   t1[18698] := -0.0536004;
   t1[18699] := -0.0617994;
   t1[18700] := 0.3399203;
   t1[18701] := 0.3337824;
   t1[18702] := 0.3265423;
   t1[18703] := 0.3181666;
   t1[18704] := 0.3086217;
   t1[18705] := 0.2978742;
   t1[18706] := 0.2858903;
   t1[18707] := 0.2726368;
   t1[18708] := 0.2580868;
   t1[18709] := 0.2423165;
   t1[18710] := 0.2254834;
   t1[18711] := 0.2077472;
   t1[18712] := 0.1892676;
   t1[18713] := 0.1702043;
   t1[18714] := 0.1507169;
   t1[18715] := 0.1309651;
   t1[18716] := 0.1111085;
   t1[18717] := 0.091307;
   t1[18718] := 0.0717201;
   t1[18719] := 0.0525076;
   t1[18720] := 0.033829;
   t1[18721] := 0.0158441;
   t1[18722] := -0.0012874;
   t1[18723] := -0.0174059;
   t1[18724] := -0.0323517;
   t1[18725] := -0.045965;
   t1[18726] := -0.0580863;
   t1[18727] := -0.0685566;
   t1[18728] := -0.0773026;
   t1[18729] := -0.084413;
   t1[18730] := -0.0899949;
   t1[18731] := -0.0941551;
   t1[18732] := -0.0970005;
   t1[18733] := -0.0986381;
   t1[18734] := -0.0991749;
   t1[18735] := -0.0987177;
   t1[18736] := -0.0973734;
   t1[18737] := -0.095249;
   t1[18738] := -0.0924515;
   t1[18739] := -0.0890877;
   t1[18740] := -0.0852646;
   t1[18741] := -0.0810891;
   t1[18742] := -0.0766682;
   t1[18743] := -0.0721086;
   t1[18744] := -0.0675175;
   t1[18745] := -0.0630017;
   t1[18746] := -0.0586682;
   t1[18747] := -0.0546078;
   t1[18748] := -0.0508318;
   t1[18749] := -0.0473261;
   t1[18750] := 0.1759748;
   t1[18751] := 0.1774203;
   t1[18752] := 0.1786771;
   t1[18753] := 0.1797362;
   t1[18754] := 0.1805886;
   t1[18755] := 0.1812253;
   t1[18756] := 0.1816373;
   t1[18757] := 0.1818157;
   t1[18758] := 0.1817521;
   t1[18759] := 0.1814474;
   t1[18760] := 0.1809096;
   t1[18761] := 0.1801469;
   t1[18762] := 0.1791678;
   t1[18763] := 0.1779805;
   t1[18764] := 0.1765932;
   t1[18765] := 0.1750143;
   t1[18766] := 0.173252;
   t1[18767] := 0.1713147;
   t1[18768] := 0.1692105;
   t1[18769] := 0.1669478;
   t1[18770] := 0.1645349;
   t1[18771] := 0.1619801;
   t1[18772] := 0.1592916;
   t1[18773] := 0.1564777;
   t1[18774] := 0.1535467;
   t1[18775] := 0.1505069;
   t1[18776] := 0.1473666;
   t1[18777] := 0.1441341;
   t1[18778] := 0.1408151;
   t1[18779] := 0.1374107;
   t1[18780] := 0.1339216;
   t1[18781] := 0.1303483;
   t1[18782] := 0.1266915;
   t1[18783] := 0.1229517;
   t1[18784] := 0.1191295;
   t1[18785] := 0.1152255;
   t1[18786] := 0.1112403;
   t1[18787] := 0.1071746;
   t1[18788] := 0.1030288;
   t1[18789] := 0.0988036;
   t1[18790] := 0.0944996;
   t1[18791] := 0.0901174;
   t1[18792] := 0.0856576;
   t1[18793] := 0.0811207;
   t1[18794] := 0.0765074;
   t1[18795] := 0.0718182;
   t1[18796] := 0.0670538;
   t1[18797] := 0.062218;
   t1[18798] := 0.057331;
   t1[18799] := 0.0524179;
   t1[18800] := 0.2070498;
   t1[18801] := 0.1995114;
   t1[18802] := 0.1919864;
   t1[18803] := 0.1845329;
   t1[18804] := 0.1772084;
   t1[18805] := 0.1700709;
   t1[18806] := 0.1631781;
   t1[18807] := 0.156588;
   t1[18808] := 0.1503544;
   t1[18809] := 0.1444713;
   t1[18810] := 0.1388855;
   t1[18811] := 0.1335424;
   t1[18812] := 0.1283877;
   t1[18813] := 0.1233668;
   t1[18814] := 0.1184252;
   t1[18815] := 0.1135085;
   t1[18816] := 0.1085621;
   t1[18817] := 0.1035315;
   t1[18818] := 0.0983623;
   t1[18819] := 0.0929999;
   t1[18820] := 0.0873899;
   t1[18821] := 0.0814778;
   t1[18822] := 0.0752091;
   t1[18823] := 0.0685292;
   t1[18824] := 0.0613837;
   t1[18825] := 0.0537182;
   t1[18826] := 0.045478;
   t1[18827] := 0.0366092;
   t1[18828] := 0.0271076;
   t1[18829] := 0.0170635;
   t1[18830] := 0.0065778;
   t1[18831] := -0.0042485;
   t1[18832] := -0.0153147;
   t1[18833] := -0.0265199;
   t1[18834] := -0.037763;
   t1[18835] := -0.0489433;
   t1[18836] := -0.0599599;
   t1[18837] := -0.0707118;
   t1[18838] := -0.0810982;
   t1[18839] := -0.0910181;
   t1[18840] := -0.1003708;
   t1[18841] := -0.1090552;
   t1[18842] := -0.1169706;
   t1[18843] := -0.124016;
   t1[18844] := -0.1300905;
   t1[18845] := -0.1350932;
   t1[18846] := -0.1389232;
   t1[18847] := -0.1415044;
   t1[18848] := -0.1428838;
   t1[18849] := -0.1431469;
   t1[18850] := 0.2326834;
   t1[18851] := 0.2246485;
   t1[18852] := 0.2165409;
   t1[18853] := 0.208421;
   t1[18854] := 0.2003494;
   t1[18855] := 0.1923865;
   t1[18856] := 0.1845929;
   t1[18857] := 0.177029;
   t1[18858] := 0.1697522;
   t1[18859] := 0.162768;
   t1[18860] := 0.1560417;
   t1[18861] := 0.1495374;
   t1[18862] := 0.1432192;
   t1[18863] := 0.1370513;
   t1[18864] := 0.1309978;
   t1[18865] := 0.1250227;
   t1[18866] := 0.1190902;
   t1[18867] := 0.1131645;
   t1[18868] := 0.1072096;
   t1[18869] := 0.1011897;
   t1[18870] := 0.0950688;
   t1[18871] := 0.0888111;
   t1[18872] := 0.0823807;
   t1[18873] := 0.0757418;
   t1[18874] := 0.0688584;
   t1[18875] := 0.0616946;
   t1[18876] := 0.0542147;
   t1[18877] := 0.0463829;
   t1[18878] := 0.0381994;
   t1[18879] := 0.0297315;
   t1[18880] := 0.0210542;
   t1[18881] := 0.0122423;
   t1[18882] := 0.0033709;
   t1[18883] := -0.0054852;
   t1[18884] := -0.014251;
   t1[18885] := -0.0228515;
   t1[18886] := -0.0312118;
   t1[18887] := -0.0392571;
   t1[18888] := -0.0469123;
   t1[18889] := -0.0541025;
   t1[18890] := -0.0607528;
   t1[18891] := -0.0667883;
   t1[18892] := -0.072134;
   t1[18893] := -0.076715;
   t1[18894] := -0.0804563;
   t1[18895] := -0.0832831;
   t1[18896] := -0.0851203;
   t1[18897] := -0.0859139;
   t1[18898] := -0.0857146;
   t1[18899] := -0.0846053;
   t1[18900] := 0.0673334;
   t1[18901] := 0.0664519;
   t1[18902] := 0.0653818;
   t1[18903] := 0.0641012;
   t1[18904] := 0.0625887;
   t1[18905] := 0.0608225;
   t1[18906] := 0.0587809;
   t1[18907] := 0.0564422;
   t1[18908] := 0.0537876;
   t1[18909] := 0.0508431;
   t1[18910] := 0.0476698;
   t1[18911] := 0.0443297;
   t1[18912] := 0.0408848;
   t1[18913] := 0.0373974;
   t1[18914] := 0.0339294;
   t1[18915] := 0.0305429;
   t1[18916] := 0.0272999;
   t1[18917] := 0.0242625;
   t1[18918] := 0.0214929;
   t1[18919] := 0.019053;
   t1[18920] := 0.0170049;
   t1[18921] := 0.0154107;
   t1[18922] := 0.0143324;
   t1[18923] := 0.0138322;
   t1[18924] := 0.013972;
   t1[18925] := 0.0148139;
   t1[18926] := 0.0164201;
   t1[18927] := 0.0188521;
   t1[18928] := 0.022123;
   t1[18929] := 0.0261538;
   t1[18930] := 0.0308553;
   t1[18931] := 0.0361382;
   t1[18932] := 0.0419132;
   t1[18933] := 0.0480911;
   t1[18934] := 0.0545826;
   t1[18935] := 0.0612985;
   t1[18936] := 0.0681495;
   t1[18937] := 0.0750462;
   t1[18938] := 0.0818996;
   t1[18939] := 0.0886203;
   t1[18940] := 0.095119;
   t1[18941] := 0.1013065;
   t1[18942] := 0.1070935;
   t1[18943] := 0.1123908;
   t1[18944] := 0.1171091;
   t1[18945] := 0.1211592;
   t1[18946] := 0.1244517;
   t1[18947] := 0.1269166;
   t1[18948] := 0.1285797;
   t1[18949] := 0.1294967;
   t1[18950] := 0.0280284;
   t1[18951] := 0.0228271;
   t1[18952] := 0.0181762;
   t1[18953] := 0.0141364;
   t1[18954] := 0.0107684;
   t1[18955] := 0.0081328;
   t1[18956] := 0.0062904;
   t1[18957] := 0.0053019;
   t1[18958] := 0.0052228;
   t1[18959] := 0.0060285;
   t1[18960] := 0.0076314;
   t1[18961] := 0.0099423;
   t1[18962] := 0.0128719;
   t1[18963] := 0.0163309;
   t1[18964] := 0.02023;
   t1[18965] := 0.0244799;
   t1[18966] := 0.0289914;
   t1[18967] := 0.0336752;
   t1[18968] := 0.0384419;
   t1[18969] := 0.0432023;
   t1[18970] := 0.0478672;
   t1[18971] := 0.0523472;
   t1[18972] := 0.056553;
   t1[18973] := 0.0603954;
   t1[18974] := 0.0637852;
   t1[18975] := 0.0666328;
   t1[18976] := 0.0688493;
   t1[18977] := 0.0703455;
   t1[18978] := 0.0710739;
   t1[18979] := 0.0710653;
   t1[18980] := 0.070359;
   t1[18981] := 0.0689945;
   t1[18982] := 0.0670113;
   t1[18983] := 0.0644488;
   t1[18984] := 0.0613464;
   t1[18985] := 0.0577437;
   t1[18986] := 0.05368;
   t1[18987] := 0.0491948;
   t1[18988] := 0.0443276;
   t1[18989] := 0.0391178;
   t1[18990] := 0.0336049;
   t1[18991] := 0.0278283;
   t1[18992] := 0.0218274;
   t1[18993] := 0.0156417;
   t1[18994] := 0.0093107;
   t1[18995] := 0.0028738;
   t1[18996] := -0.0036295;
   t1[18997] := -0.0101605;
   t1[18998] := -0.0166832;
   t1[18999] := -0.0231627;
   t1[19000] := 0.0320975;
   t1[19001] := 0.0306463;
   t1[19002] := 0.0295504;
   t1[19003] := 0.0288107;
   t1[19004] := 0.0284277;
   t1[19005] := 0.0284023;
   t1[19006] := 0.028735;
   t1[19007] := 0.0294266;
   t1[19008] := 0.0304775;
   t1[19009] := 0.0318814;
   t1[19010] := 0.0336268;
   t1[19011] := 0.0357022;
   t1[19012] := 0.0380961;
   t1[19013] := 0.0407971;
   t1[19014] := 0.0437935;
   t1[19015] := 0.0470737;
   t1[19016] := 0.0506264;
   t1[19017] := 0.0544399;
   t1[19018] := 0.0585028;
   t1[19019] := 0.0628034;
   t1[19020] := 0.0673303;
   t1[19021] := 0.0720719;
   t1[19022] := 0.0770167;
   t1[19023] := 0.0821532;
   t1[19024] := 0.0874698;
   t1[19025] := 0.092955;
   t1[19026] := 0.0985973;
   t1[19027] := 0.104385;
   t1[19028] := 0.1102992;
   t1[19029] := 0.1163065;
   t1[19030] := 0.1223722;
   t1[19031] := 0.1284615;
   t1[19032] := 0.1345395;
   t1[19033] := 0.1405715;
   t1[19034] := 0.1465226;
   t1[19035] := 0.1523581;
   t1[19036] := 0.1580431;
   t1[19037] := 0.1635428;
   t1[19038] := 0.1688224;
   t1[19039] := 0.1738472;
   t1[19040] := 0.1785823;
   t1[19041] := 0.1829928;
   t1[19042] := 0.1870441;
   t1[19043] := 0.1907013;
   t1[19044] := 0.1939295;
   t1[19045] := 0.196694;
   t1[19046] := 0.1989601;
   t1[19047] := 0.2006966;
   t1[19048] := 0.2018923;
   t1[19049] := 0.2025419;
   t1[19050] := 0.3164727;
   t1[19051] := 0.3206323;
   t1[19052] := 0.3240848;
   t1[19053] := 0.3267758;
   t1[19054] := 0.3286505;
   t1[19055] := 0.3296546;
   t1[19056] := 0.3297334;
   t1[19057] := 0.3288324;
   t1[19058] := 0.3269007;
   t1[19059] := 0.3239454;
   t1[19060] := 0.3200189;
   t1[19061] := 0.3151748;
   t1[19062] := 0.3094669;
   t1[19063] := 0.3029487;
   t1[19064] := 0.2956739;
   t1[19065] := 0.2876963;
   t1[19066] := 0.2790695;
   t1[19067] := 0.2698471;
   t1[19068] := 0.2600828;
   t1[19069] := 0.2498303;
   t1[19070] := 0.2391432;
   t1[19071] := 0.2280753;
   t1[19072] := 0.2166801;
   t1[19073] := 0.2050114;
   t1[19074] := 0.1931227;
   t1[19075] := 0.1810679;
   t1[19076] := 0.1689004;
   t1[19077] := 0.1566742;
   t1[19078] := 0.1444511;
   t1[19079] := 0.1323085;
   t1[19080] := 0.1203256;
   t1[19081] := 0.1085816;
   t1[19082] := 0.0971556;
   t1[19083] := 0.0861267;
   t1[19084] := 0.0755742;
   t1[19085] := 0.0655772;
   t1[19086] := 0.0562149;
   t1[19087] := 0.0475663;
   t1[19088] := 0.0397108;
   t1[19089] := 0.0327274;
   t1[19090] := 0.0266954;
   t1[19091] := 0.0216937;
   t1[19092] := 0.0178018;
   t1[19093] := 0.0150986;
   t1[19094] := 0.0136634;
   t1[19095] := 0.0135753;
   t1[19096] := 0.0149134;
   t1[19097] := 0.0177261;
   t1[19098] := 0.0219068;
   t1[19099] := 0.0273009;
   t1[19100] := 0.0081115;
   t1[19101] := 0.0047921;
   t1[19102] := 0.0018571;
   t1[19103] := -0.0006861;
   t1[19104] := -0.0028299;
   t1[19105] := -0.0045669;
   t1[19106] := -0.0058896;
   t1[19107] := -0.0067905;
   t1[19108] := -0.0072618;
   t1[19109] := -0.0072895;
   t1[19110] := -0.0068552;
   t1[19111] := -0.00594;
   t1[19112] := -0.0045253;
   t1[19113] := -0.0025923;
   t1[19114] := -0.0001223;
   t1[19115] := 0.0029033;
   t1[19116] := 0.0065034;
   t1[19117] := 0.0106967;
   t1[19118] := 0.0155018;
   t1[19119] := 0.0209374;
   t1[19120] := 0.0270224;
   t1[19121] := 0.0337754;
   t1[19122] := 0.0412151;
   t1[19123] := 0.0493603;
   t1[19124] := 0.0582296;
   t1[19125] := 0.0678419;
   t1[19126] := 0.0782157;
   t1[19127] := 0.0893694;
   t1[19128] := 0.1012631;
   t1[19129] := 0.1137472;
   t1[19130] := 0.1266599;
   t1[19131] := 0.139839;
   t1[19132] := 0.1531228;
   t1[19133] := 0.1663493;
   t1[19134] := 0.1793567;
   t1[19135] := 0.1919829;
   t1[19136] := 0.204066;
   t1[19137] := 0.2154442;
   t1[19138] := 0.2259555;
   t1[19139] := 0.2354381;
   t1[19140] := 0.2437299;
   t1[19141] := 0.250669;
   t1[19142] := 0.2560937;
   t1[19143] := 0.2598418;
   t1[19144] := 0.2617516;
   t1[19145] := 0.261661;
   t1[19146] := 0.2594082;
   t1[19147] := 0.2548787;
   t1[19148] := 0.248195;
   t1[19149] := 0.2395535;
   t1[19150] := 0.3116351;
   t1[19151] := 0.3118189;
   t1[19152] := 0.311274;
   t1[19153] := 0.30992;
   t1[19154] := 0.3076764;
   t1[19155] := 0.3044629;
   t1[19156] := 0.3001987;
   t1[19157] := 0.2948037;
   t1[19158] := 0.2882029;
   t1[19159] := 0.2804078;
   t1[19160] := 0.271498;
   t1[19161] := 0.2615548;
   t1[19162] := 0.2506597;
   t1[19163] := 0.238894;
   t1[19164] := 0.2263391;
   t1[19165] := 0.2130764;
   t1[19166] := 0.1991872;
   t1[19167] := 0.184753;
   t1[19168] := 0.1698552;
   t1[19169] := 0.1545751;
   t1[19170] := 0.1389941;
   t1[19171] := 0.1231935;
   t1[19172] := 0.1072549;
   t1[19173] := 0.0912595;
   t1[19174] := 0.0752887;
   t1[19175] := 0.059424;
   t1[19176] := 0.0437467;
   t1[19177] := 0.0283381;
   t1[19178] := 0.0132743;
   t1[19179] := -0.0013792;
   t1[19180] := -0.0155577;
   t1[19181] := -0.0291967;
   t1[19182] := -0.0422315;
   t1[19183] := -0.0545976;
   t1[19184] := -0.0662306;
   t1[19185] := -0.0770656;
   t1[19186] := -0.0870383;
   t1[19187] := -0.0960839;
   t1[19188] := -0.104138;
   t1[19189] := -0.1111361;
   t1[19190] := -0.1170134;
   t1[19191] := -0.1217054;
   t1[19192] := -0.1251476;
   t1[19193] := -0.1272754;
   t1[19194] := -0.1280243;
   t1[19195] := -0.1273295;
   t1[19196] := -0.1251266;
   t1[19197] := -0.1213727;
   t1[19198] := -0.1161325;
   t1[19199] := -0.1095048;
   t1[19200] := 0.031007;
   t1[19201] := 0.0430812;
   t1[19202] := 0.0550985;
   t1[19203] := 0.0669886;
   t1[19204] := 0.0786809;
   t1[19205] := 0.0901053;
   t1[19206] := 0.1011912;
   t1[19207] := 0.1118682;
   t1[19208] := 0.1220685;
   t1[19209] := 0.1317644;
   t1[19210] := 0.1409596;
   t1[19211] := 0.1496588;
   t1[19212] := 0.1578664;
   t1[19213] := 0.1655871;
   t1[19214] := 0.1728256;
   t1[19215] := 0.1795864;
   t1[19216] := 0.1858741;
   t1[19217] := 0.1916933;
   t1[19218] := 0.1970486;
   t1[19219] := 0.2019446;
   t1[19220] := 0.206386;
   t1[19221] := 0.2103773;
   t1[19222] := 0.2139231;
   t1[19223] := 0.2170281;
   t1[19224] := 0.2196967;
   t1[19225] := 0.2219336;
   t1[19226] := 0.2237435;
   t1[19227] := 0.2251309;
   t1[19228] := 0.226105;
   t1[19229] := 0.2266827;
   t1[19230] := 0.2268822;
   t1[19231] := 0.2267217;
   t1[19232] := 0.2262192;
   t1[19233] := 0.2253929;
   t1[19234] := 0.2242608;
   t1[19235] := 0.2228411;
   t1[19236] := 0.2211518;
   t1[19237] := 0.2192111;
   t1[19238] := 0.2170371;
   t1[19239] := 0.2146478;
   t1[19240] := 0.2120615;
   t1[19241] := 0.2092961;
   t1[19242] := 0.2063698;
   t1[19243] := 0.2033007;
   t1[19244] := 0.2001069;
   t1[19245] := 0.1968066;
   t1[19246] := 0.1934177;
   t1[19247] := 0.1899561;
   t1[19248] := 0.186425;
   t1[19249] := 0.182824;
   t1[19250] := -0.0120644;
   t1[19251] := 0.001842;
   t1[19252] := 0.0152882;
   t1[19253] := 0.0281604;
   t1[19254] := 0.040345;
   t1[19255] := 0.0517284;
   t1[19256] := 0.0621967;
   t1[19257] := 0.0716364;
   t1[19258] := 0.0799405;
   t1[19259] := 0.0871045;
   t1[19260] := 0.0932047;
   t1[19261] := 0.0983197;
   t1[19262] := 0.102528;
   t1[19263] := 0.1059081;
   t1[19264] := 0.1085385;
   t1[19265] := 0.1104977;
   t1[19266] := 0.1118644;
   t1[19267] := 0.1127169;
   t1[19268] := 0.1131338;
   t1[19269] := 0.1131936;
   t1[19270] := 0.1129749;
   t1[19271] := 0.1125562;
   t1[19272] := 0.1120159;
   t1[19273] := 0.1114327;
   t1[19274] := 0.1108849;
   t1[19275] := 0.1104512;
   t1[19276] := 0.1102101;
   t1[19277] := 0.1102396;
   t1[19278] := 0.1105719;
   t1[19279] := 0.1111515;
   t1[19280] := 0.1119133;
   t1[19281] := 0.1127922;
   t1[19282] := 0.1137231;
   t1[19283] := 0.1146409;
   t1[19284] := 0.1154805;
   t1[19285] := 0.1161768;
   t1[19286] := 0.1166647;
   t1[19287] := 0.116879;
   t1[19288] := 0.1167547;
   t1[19289] := 0.1162266;
   t1[19290] := 0.1152296;
   t1[19291] := 0.1136987;
   t1[19292] := 0.1115686;
   t1[19293] := 0.1087744;
   t1[19294] := 0.1052508;
   t1[19295] := 0.1009329;
   t1[19296] := 0.0957554;
   t1[19297] := 0.0896758;
   t1[19298] := 0.0827645;
   t1[19299] := 0.0751271;
   t1[19300] := 0.1167602;
   t1[19301] := 0.1285919;
   t1[19302] := 0.1400018;
   t1[19303] := 0.1508942;
   t1[19304] := 0.1611734;
   t1[19305] := 0.1707437;
   t1[19306] := 0.1795094;
   t1[19307] := 0.1873749;
   t1[19308] := 0.1942492;
   t1[19309] := 0.2001155;
   t1[19310] := 0.2050154;
   t1[19311] := 0.2089921;
   t1[19312] := 0.2120888;
   t1[19313] := 0.2143485;
   t1[19314] := 0.2158144;
   t1[19315] := 0.2165298;
   t1[19316] := 0.2165377;
   t1[19317] := 0.2158812;
   t1[19318] := 0.2146037;
   t1[19319] := 0.2127481;
   t1[19320] := 0.2103577;
   t1[19321] := 0.2074756;
   t1[19322] := 0.204145;
   t1[19323] := 0.200409;
   t1[19324] := 0.1963107;
   t1[19325] := 0.1918934;
   t1[19326] := 0.1872001;
   t1[19327] := 0.182274;
   t1[19328] := 0.1771547;
   t1[19329] := 0.1718746;
   t1[19330] := 0.1664655;
   t1[19331] := 0.1609593;
   t1[19332] := 0.1553877;
   t1[19333] := 0.1497826;
   t1[19334] := 0.1441758;
   t1[19335] := 0.138599;
   t1[19336] := 0.133084;
   t1[19337] := 0.1276627;
   t1[19338] := 0.1223669;
   t1[19339] := 0.1172283;
   t1[19340] := 0.1122788;
   t1[19341] := 0.1075501;
   t1[19342] := 0.1030742;
   t1[19343] := 0.0988826;
   t1[19344] := 0.0950073;
   t1[19345] := 0.0914801;
   t1[19346] := 0.0883328;
   t1[19347] := 0.0855882;
   t1[19348] := 0.0832247;
   t1[19349] := 0.0812067;
   t1[19350] := 0.2197201;
   t1[19351] := 0.2172861;
   t1[19352] := 0.2143028;
   t1[19353] := 0.2107741;
   t1[19354] := 0.2067038;
   t1[19355] := 0.2020957;
   t1[19356] := 0.1969537;
   t1[19357] := 0.1912815;
   t1[19358] := 0.1850853;
   t1[19359] := 0.1784045;
   t1[19360] := 0.1713053;
   t1[19361] := 0.1638544;
   t1[19362] := 0.1561187;
   t1[19363] := 0.1481647;
   t1[19364] := 0.1400594;
   t1[19365] := 0.1318695;
   t1[19366] := 0.1236617;
   t1[19367] := 0.1155029;
   t1[19368] := 0.1074598;
   t1[19369] := 0.0995992;
   t1[19370] := 0.0919878;
   t1[19371] := 0.0846924;
   t1[19372] := 0.0777798;
   t1[19373] := 0.0713168;
   t1[19374] := 0.06537;
   t1[19375] := 0.0600064;
   t1[19376] := 0.0552926;
   t1[19377] := 0.051295;
   t1[19378] := 0.0480385;
   t1[19379] := 0.0454686;
   t1[19380] := 0.0435222;
   t1[19381] := 0.0421363;
   t1[19382] := 0.0412477;
   t1[19383] := 0.0407934;
   t1[19384] := 0.04071;
   t1[19385] := 0.0409347;
   t1[19386] := 0.0414042;
   t1[19387] := 0.0420554;
   t1[19388] := 0.0428252;
   t1[19389] := 0.0436506;
   t1[19390] := 0.0444683;
   t1[19391] := 0.0452152;
   t1[19392] := 0.0458283;
   t1[19393] := 0.0462444;
   t1[19394] := 0.0464004;
   t1[19395] := 0.0462332;
   t1[19396] := 0.0456796;
   t1[19397] := 0.0446904;
   t1[19398] := 0.0432853;
   t1[19399] := 0.0415054;
   t1[19400] := -0.0723167;
   t1[19401] := -0.0811981;
   t1[19402] := -0.0889529;
   t1[19403] := -0.0955175;
   t1[19404] := -0.1008282;
   t1[19405] := -0.1048214;
   t1[19406] := -0.1074335;
   t1[19407] := -0.1086009;
   t1[19408] := -0.1082657;
   t1[19409] := -0.1064598;
   t1[19410] := -0.103286;
   t1[19411] := -0.0988486;
   t1[19412] := -0.0932522;
   t1[19413] := -0.0866013;
   t1[19414] := -0.0790003;
   t1[19415] := -0.0705539;
   t1[19416] := -0.0613663;
   t1[19417] := -0.0515423;
   t1[19418] := -0.0411863;
   t1[19419] := -0.0304028;
   t1[19420] := -0.0192962;
   t1[19421] := -0.0079711;
   t1[19422] := 0.003468;
   t1[19423] := 0.0149166;
   t1[19424] := 0.0262703;
   t1[19425] := 0.0374244;
   t1[19426] := 0.0482745;
   t1[19427] := 0.0587165;
   t1[19428] := 0.0686813;
   t1[19429] := 0.0781667;
   t1[19430] := 0.087178;
   t1[19431] := 0.0957204;
   t1[19432] := 0.1037991;
   t1[19433] := 0.1114193;
   t1[19434] := 0.1185863;
   t1[19435] := 0.1253053;
   t1[19436] := 0.1315816;
   t1[19437] := 0.1374203;
   t1[19438] := 0.1428267;
   t1[19439] := 0.147806;
   t1[19440] := 0.1523635;
   t1[19441] := 0.1565043;
   t1[19442] := 0.1602338;
   t1[19443] := 0.1635571;
   t1[19444] := 0.1664795;
   t1[19445] := 0.1690062;
   t1[19446] := 0.1711424;
   t1[19447] := 0.1728936;
   t1[19448] := 0.1742667;
   t1[19449] := 0.1752688;
   t1[19450] := 0.0910374;
   t1[19451] := 0.0981503;
   t1[19452] := 0.1054753;
   t1[19453] := 0.1130103;
   t1[19454] := 0.120753;
   t1[19455] := 0.1287014;
   t1[19456] := 0.1368533;
   t1[19457] := 0.1452066;
   t1[19458] := 0.1537566;
   t1[19459] := 0.1624598;
   t1[19460] := 0.1712421;
   t1[19461] := 0.1800283;
   t1[19462] := 0.1887436;
   t1[19463] := 0.1973128;
   t1[19464] := 0.2056611;
   t1[19465] := 0.2137134;
   t1[19466] := 0.2213947;
   t1[19467] := 0.2286299;
   t1[19468] := 0.2353442;
   t1[19469] := 0.2414626;
   t1[19470] := 0.2469099;
   t1[19471] := 0.2516112;
   t1[19472] := 0.2554916;
   t1[19473] := 0.2584759;
   t1[19474] := 0.2604892;
   t1[19475] := 0.2614565;
   t1[19476] := 0.2613029;
   t1[19477] := 0.2599536;
   t1[19478] := 0.2573789;
   t1[19479] := 0.2536334;
   t1[19480] := 0.2487813;
   t1[19481] := 0.2428869;
   t1[19482] := 0.2360145;
   t1[19483] := 0.2282281;
   t1[19484] := 0.219592;
   t1[19485] := 0.2101706;
   t1[19486] := 0.2000278;
   t1[19487] := 0.1892281;
   t1[19488] := 0.1778356;
   t1[19489] := 0.1659145;
   t1[19490] := 0.153529;
   t1[19491] := 0.1407434;
   t1[19492] := 0.127622;
   t1[19493] := 0.1142288;
   t1[19494] := 0.1006281;
   t1[19495] := 0.0868841;
   t1[19496] := 0.0730612;
   t1[19497] := 0.0592237;
   t1[19498] := 0.0454382;
   t1[19499] := 0.0317715;
   t1[19500] := 0.1190348;
   t1[19501] := 0.1201077;
   t1[19502] := 0.1206658;
   t1[19503] := 0.1206494;
   t1[19504] := 0.119999;
   t1[19505] := 0.1186547;
   t1[19506] := 0.1165569;
   t1[19507] := 0.113646;
   t1[19508] := 0.1098679;
   t1[19509] := 0.1052543;
   t1[19510] := 0.0999048;
   t1[19511] := 0.0939205;
   t1[19512] := 0.0874028;
   t1[19513] := 0.0804529;
   t1[19514] := 0.0731721;
   t1[19515] := 0.0656616;
   t1[19516] := 0.0580227;
   t1[19517] := 0.0503567;
   t1[19518] := 0.0427649;
   t1[19519] := 0.0353485;
   t1[19520] := 0.0282087;
   t1[19521] := 0.0214469;
   t1[19522] := 0.0151643;
   t1[19523] := 0.0094621;
   t1[19524] := 0.0044417;
   t1[19525] := 0.0002044;
   t1[19526] := -0.0031487;
   t1[19527] := -0.0055168;
   t1[19528] := -0.0068551;
   t1[19529] := -0.007225;
   t1[19530] := -0.0066997;
   t1[19531] := -0.0053527;
   t1[19532] := -0.0032571;
   t1[19533] := -0.0004863;
   t1[19534] := 0.0028866;
   t1[19535] := 0.0067881;
   t1[19536] := 0.0111451;
   t1[19537] := 0.0158843;
   t1[19538] := 0.0209324;
   t1[19539] := 0.026216;
   t1[19540] := 0.0316621;
   t1[19541] := 0.0371971;
   t1[19542] := 0.042748;
   t1[19543] := 0.0482413;
   t1[19544] := 0.0536039;
   t1[19545] := 0.0587625;
   t1[19546] := 0.0636437;
   t1[19547] := 0.068184;
   t1[19548] := 0.0723681;
   t1[19549] := 0.0761959;
   t1[19550] := -0.0686139;
   t1[19551] := -0.0550236;
   t1[19552] := -0.0416787;
   t1[19553] := -0.0286607;
   t1[19554] := -0.0160508;
   t1[19555] := -0.0039303;
   t1[19556] := 0.0076195;
   t1[19557] := 0.0185172;
   t1[19558] := 0.0286869;
   t1[19559] := 0.0381341;
   t1[19560] := 0.0469288;
   t1[19561] := 0.0551423;
   t1[19562] := 0.0628465;
   t1[19563] := 0.0701128;
   t1[19564] := 0.0770127;
   t1[19565] := 0.083618;
   t1[19566] := 0.0900002;
   t1[19567] := 0.0962308;
   t1[19568] := 0.1023815;
   t1[19569] := 0.1085237;
   t1[19570] := 0.1147292;
   t1[19571] := 0.1210695;
   t1[19572] := 0.1276161;
   t1[19573] := 0.1344407;
   t1[19574] := 0.1416148;
   t1[19575] := 0.1492099;
   t1[19576] := 0.1572978;
   t1[19577] := 0.1659495;
   t1[19578] := 0.1751826;
   t1[19579] := 0.1849134;
   t1[19580] := 0.1950468;
   t1[19581] := 0.2054878;
   t1[19582] := 0.2161414;
   t1[19583] := 0.2269125;
   t1[19584] := 0.237706;
   t1[19585] := 0.2484269;
   t1[19586] := 0.2589802;
   t1[19587] := 0.2692708;
   t1[19588] := 0.2792036;
   t1[19589] := 0.2886837;
   t1[19590] := 0.2976158;
   t1[19591] := 0.3059051;
   t1[19592] := 0.3134564;
   t1[19593] := 0.3201748;
   t1[19594] := 0.3259652;
   t1[19595] := 0.3307323;
   t1[19596] := 0.3343814;
   t1[19597] := 0.3368372;
   t1[19598] := 0.3381237;
   t1[19599] := 0.3382958;
   t1[19600] := -0.0348268;
   t1[19601] := -0.0426686;
   t1[19602] := -0.050124;
   t1[19603] := -0.0571507;
   t1[19604] := -0.0637064;
   t1[19605] := -0.0697488;
   t1[19606] := -0.0752356;
   t1[19607] := -0.0801245;
   t1[19608] := -0.0843756;
   t1[19609] := -0.0879853;
   t1[19610] := -0.0909789;
   t1[19611] := -0.0933823;
   t1[19612] := -0.0952214;
   t1[19613] := -0.0965222;
   t1[19614] := -0.0973106;
   t1[19615] := -0.0976127;
   t1[19616] := -0.0974543;
   t1[19617] := -0.0968613;
   t1[19618] := -0.0958598;
   t1[19619] := -0.0944757;
   t1[19620] := -0.0927349;
   t1[19621] := -0.0906634;
   t1[19622] := -0.0882871;
   t1[19623] := -0.085632;
   t1[19624] := -0.0827241;
   t1[19625] := -0.0795892;
   t1[19626] := -0.0762534;
   t1[19627] := -0.0727425;
   t1[19628] := -0.069084;
   t1[19629] := -0.0653077;
   t1[19630] := -0.0614438;
   t1[19631] := -0.0575227;
   t1[19632] := -0.0535745;
   t1[19633] := -0.0496293;
   t1[19634] := -0.0457175;
   t1[19635] := -0.0418693;
   t1[19636] := -0.0381148;
   t1[19637] := -0.0344843;
   t1[19638] := -0.031008;
   t1[19639] := -0.0277162;
   t1[19640] := -0.024639;
   t1[19641] := -0.0218066;
   t1[19642] := -0.0192493;
   t1[19643] := -0.0169972;
   t1[19644] := -0.0150807;
   t1[19645] := -0.0135299;
   t1[19646] := -0.0123751;
   t1[19647] := -0.011637;
   t1[19648] := -0.0112897;
   t1[19649] := -0.0112926;
   t1[19650] := 0.1051766;
   t1[19651] := 0.1102797;
   t1[19652] := 0.1147799;
   t1[19653] := 0.1185808;
   t1[19654] := 0.1215865;
   t1[19655] := 0.1237005;
   t1[19656] := 0.1248267;
   t1[19657] := 0.1248689;
   t1[19658] := 0.1237374;
   t1[19659] := 0.121445;
   t1[19660] := 0.1180852;
   t1[19661] := 0.1137535;
   t1[19662] := 0.1085456;
   t1[19663] := 0.102557;
   t1[19664] := 0.0958833;
   t1[19665] := 0.0886201;
   t1[19666] := 0.080863;
   t1[19667] := 0.0727076;
   t1[19668] := 0.0642495;
   t1[19669] := 0.0555842;
   t1[19670] := 0.0468074;
   t1[19671] := 0.0380146;
   t1[19672] := 0.0293015;
   t1[19673] := 0.0207636;
   t1[19674] := 0.0124965;
   t1[19675] := 0.0045958;
   t1[19676] := -0.0028428;
   t1[19677] := -0.0097242;
   t1[19678] := -0.0159896;
   t1[19679] := -0.0216493;
   t1[19680] := -0.0267216;
   t1[19681] := -0.0312245;
   t1[19682] := -0.0351762;
   t1[19683] := -0.0385948;
   t1[19684] := -0.0414984;
   t1[19685] := -0.0439053;
   t1[19686] := -0.0458334;
   t1[19687] := -0.047301;
   t1[19688] := -0.0483262;
   t1[19689] := -0.0489271;
   t1[19690] := -0.0491219;
   t1[19691] := -0.0489287;
   t1[19692] := -0.0483656;
   t1[19693] := -0.0474507;
   t1[19694] := -0.0462023;
   t1[19695] := -0.0446384;
   t1[19696] := -0.0427772;
   t1[19697] := -0.040637;
   t1[19698] := -0.0382374;
   t1[19699] := -0.0355984;
   t1[19700] := 0.117127;
   t1[19701] := 0.1166275;
   t1[19702] := 0.1160149;
   t1[19703] := 0.115284;
   t1[19704] := 0.1144297;
   t1[19705] := 0.1134468;
   t1[19706] := 0.1123303;
   t1[19707] := 0.111075;
   t1[19708] := 0.1096755;
   t1[19709] := 0.1081229;
   t1[19710] := 0.106405;
   t1[19711] := 0.1045097;
   t1[19712] := 0.1024249;
   t1[19713] := 0.1001385;
   t1[19714] := 0.0976384;
   t1[19715] := 0.0949125;
   t1[19716] := 0.0919486;
   t1[19717] := 0.0887347;
   t1[19718] := 0.0852586;
   t1[19719] := 0.0815083;
   t1[19720] := 0.0774716;
   t1[19721] := 0.0731363;
   t1[19722] := 0.0684905;
   t1[19723] := 0.0635219;
   t1[19724] := 0.0582185;
   t1[19725] := 0.0525682;
   t1[19726] := 0.0465587;
   t1[19727] := 0.0401784;
   t1[19728] := 0.033439;
   t1[19729] := 0.0263979;
   t1[19730] := 0.0191174;
   t1[19731] := 0.0116598;
   t1[19732] := 0.0040874;
   t1[19733] := -0.0035376;
   t1[19734] := -0.0111528;
   t1[19735] := -0.0186958;
   t1[19736] := -0.0261045;
   t1[19737] := -0.0333164;
   t1[19738] := -0.0402694;
   t1[19739] := -0.046901;
   t1[19740] := -0.053149;
   t1[19741] := -0.058951;
   t1[19742] := -0.0642449;
   t1[19743] := -0.0689682;
   t1[19744] := -0.0730587;
   t1[19745] := -0.076454;
   t1[19746] := -0.0790919;
   t1[19747] := -0.080925;
   t1[19748] := -0.0819811;
   t1[19749] := -0.0823112;
   t1[19750] := 0.0605384;
   t1[19751] := 0.0596309;
   t1[19752] := 0.0589958;
   t1[19753] := 0.0586726;
   t1[19754] := 0.0587013;
   t1[19755] := 0.0591213;
   t1[19756] := 0.0599725;
   t1[19757] := 0.0612945;
   t1[19758] := 0.063123;
   t1[19759] := 0.0654314;
   t1[19760] := 0.0681442;
   t1[19761] := 0.0711845;
   t1[19762] := 0.0744753;
   t1[19763] := 0.0779398;
   t1[19764] := 0.081501;
   t1[19765] := 0.0850821;
   t1[19766] := 0.0886061;
   t1[19767] := 0.0919962;
   t1[19768] := 0.0951755;
   t1[19769] := 0.0980671;
   t1[19770] := 0.100594;
   t1[19771] := 0.1026793;
   t1[19772] := 0.1042462;
   t1[19773] := 0.1052178;
   t1[19774] := 0.1055172;
   t1[19775] := 0.1050674;
   t1[19776] := 0.1037916;
   t1[19777] := 0.1016133;
   t1[19778] := 0.0985063;
   t1[19779] := 0.0945396;
   t1[19780] := 0.089793;
   t1[19781] := 0.084346;
   t1[19782] := 0.0782784;
   t1[19783] := 0.0716697;
   t1[19784] := 0.0645998;
   t1[19785] := 0.0571482;
   t1[19786] := 0.0493947;
   t1[19787] := 0.0414188;
   t1[19788] := 0.0333003;
   t1[19789] := 0.0251189;
   t1[19790] := 0.0169541;
   t1[19791] := 0.0088857;
   t1[19792] := 0.0009933;
   t1[19793] := -0.0066434;
   t1[19794] := -0.0139447;
   t1[19795] := -0.0208309;
   t1[19796] := -0.0272225;
   t1[19797] := -0.033052;
   t1[19798] := -0.038314;
   t1[19799] := -0.0430221;
   t1[19800] := 0.0497248;
   t1[19801] := 0.0548617;
   t1[19802] := 0.0597544;
   t1[19803] := 0.0643751;
   t1[19804] := 0.0686959;
   t1[19805] := 0.0726891;
   t1[19806] := 0.0763267;
   t1[19807] := 0.0795811;
   t1[19808] := 0.0824267;
   t1[19809] := 0.0848719;
   t1[19810] := 0.0869523;
   t1[19811] := 0.0887043;
   t1[19812] := 0.090164;
   t1[19813] := 0.0913678;
   t1[19814] := 0.0923519;
   t1[19815] := 0.0931525;
   t1[19816] := 0.093806;
   t1[19817] := 0.0943485;
   t1[19818] := 0.0948164;
   t1[19819] := 0.0952459;
   t1[19820] := 0.0956733;
   t1[19821] := 0.0961348;
   t1[19822] := 0.0966667;
   t1[19823] := 0.0973053;
   t1[19824] := 0.0980867;
   t1[19825] := 0.0990474;
   t1[19826] := 0.1002235;
   t1[19827] := 0.101651;
   t1[19828] := 0.1033362;
   t1[19829] := 0.1052285;
   t1[19830] := 0.1072712;
   t1[19831] := 0.1094076;
   t1[19832] := 0.111581;
   t1[19833] := 0.1137345;
   t1[19834] := 0.1158115;
   t1[19835] := 0.1177552;
   t1[19836] := 0.1195088;
   t1[19837] := 0.1210157;
   t1[19838] := 0.122219;
   t1[19839] := 0.123062;
   t1[19840] := 0.123488;
   t1[19841] := 0.1234403;
   t1[19842] := 0.122862;
   t1[19843] := 0.1216965;
   t1[19844] := 0.119887;
   t1[19845] := 0.1173768;
   t1[19846] := 0.1141091;
   t1[19847] := 0.1100459;
   t1[19848] := 0.1052429;
   t1[19849] := 0.0997852;
   t1[19850] := 0.1509402;
   t1[19851] := 0.1470928;
   t1[19852] := 0.1432999;
   t1[19853] := 0.1396035;
   t1[19854] := 0.1360461;
   t1[19855] := 0.1326696;
   t1[19856] := 0.1295165;
   t1[19857] := 0.1266288;
   t1[19858] := 0.1240469;
   t1[19859] := 0.1217828;
   t1[19860] := 0.119826;
   t1[19861] := 0.1181654;
   t1[19862] := 0.1167899;
   t1[19863] := 0.1156884;
   t1[19864] := 0.1148499;
   t1[19865] := 0.1142632;
   t1[19866] := 0.1139174;
   t1[19867] := 0.1138012;
   t1[19868] := 0.1139036;
   t1[19869] := 0.1142136;
   t1[19870] := 0.1147201;
   t1[19871] := 0.1154119;
   t1[19872] := 0.116278;
   t1[19873] := 0.1173073;
   t1[19874] := 0.1184887;
   t1[19875] := 0.1198112;
   t1[19876] := 0.1212636;
   t1[19877] := 0.1228348;
   t1[19878] := 0.124502;
   t1[19879] := 0.1262204;
   t1[19880] := 0.127943;
   t1[19881] := 0.1296225;
   t1[19882] := 0.1312117;
   t1[19883] := 0.1326635;
   t1[19884] := 0.1339306;
   t1[19885] := 0.134966;
   t1[19886] := 0.1357223;
   t1[19887] := 0.1361525;
   t1[19888] := 0.1362094;
   t1[19889] := 0.1358457;
   t1[19890] := 0.1350143;
   t1[19891] := 0.1336681;
   t1[19892] := 0.1317597;
   t1[19893] := 0.1292422;
   t1[19894] := 0.1260682;
   t1[19895] := 0.1221906;
   t1[19896] := 0.1175622;
   t1[19897] := 0.1121553;
   t1[19898] := 0.1060389;
   t1[19899] := 0.0993124;
   t1[19900] := 0.1816427;
   t1[19901] := 0.1859255;
   t1[19902] := 0.1899239;
   t1[19903] := 0.1936141;
   t1[19904] := 0.1969721;
   t1[19905] := 0.1999743;
   t1[19906] := 0.2025966;
   t1[19907] := 0.2048154;
   t1[19908] := 0.2066072;
   t1[19909] := 0.2079562;
   t1[19910] := 0.2088525;
   t1[19911] := 0.2092866;
   t1[19912] := 0.2092486;
   t1[19913] := 0.2087289;
   t1[19914] := 0.2077178;
   t1[19915] := 0.2062056;
   t1[19916] := 0.2041826;
   t1[19917] := 0.2016391;
   t1[19918] := 0.1985655;
   t1[19919] := 0.194952;
   t1[19920] := 0.1907889;
   t1[19921] := 0.1860666;
   t1[19922] := 0.1807753;
   t1[19923] := 0.1749054;
   t1[19924] := 0.1684471;
   t1[19925] := 0.1613909;
   t1[19926] := 0.1537269;
   t1[19927] := 0.1454457;
   t1[19928] := 0.1365594;
   t1[19929] := 0.127121;
   t1[19930] := 0.117188;
   t1[19931] := 0.1068182;
   t1[19932] := 0.0960691;
   t1[19933] := 0.0849982;
   t1[19934] := 0.0736632;
   t1[19935] := 0.0621217;
   t1[19936] := 0.0504312;
   t1[19937] := 0.0386494;
   t1[19938] := 0.0268339;
   t1[19939] := 0.0150421;
   t1[19940] := 0.0033319;
   t1[19941] := -0.0082393;
   t1[19942] := -0.0196139;
   t1[19943] := -0.0307344;
   t1[19944] := -0.0415429;
   t1[19945] := -0.0519821;
   t1[19946] := -0.0619942;
   t1[19947] := -0.071527;
   t1[19948] := -0.0805537;
   t1[19949] := -0.089056;
   t1[19950] := 0.0638854;
   t1[19951] := 0.0717888;
   t1[19952] := 0.0798736;
   t1[19953] := 0.0880734;
   t1[19954] := 0.0963217;
   t1[19955] := 0.1045522;
   t1[19956] := 0.1126982;
   t1[19957] := 0.1206934;
   t1[19958] := 0.1284724;
   t1[19959] := 0.1359862;
   t1[19960] := 0.1431986;
   t1[19961] := 0.1500738;
   t1[19962] := 0.1565761;
   t1[19963] := 0.1626695;
   t1[19964] := 0.1683184;
   t1[19965] := 0.1734868;
   t1[19966] := 0.1781391;
   t1[19967] := 0.1822393;
   t1[19968] := 0.1857518;
   t1[19969] := 0.1886406;
   t1[19970] := 0.19087;
   t1[19971] := 0.1924042;
   t1[19972] := 0.1932074;
   t1[19973] := 0.1932438;
   t1[19974] := 0.1924774;
   t1[19975] := 0.1908727;
   t1[19976] := 0.1883938;
   t1[19977] := 0.1850051;
   t1[19978] := 0.1807017;
   t1[19979] := 0.1755369;
   t1[19980] := 0.1695705;
   t1[19981] := 0.162862;
   t1[19982] := 0.1554713;
   t1[19983] := 0.147458;
   t1[19984] := 0.1388818;
   t1[19985] := 0.1298026;
   t1[19986] := 0.1202799;
   t1[19987] := 0.1103736;
   t1[19988] := 0.1001432;
   t1[19989] := 0.0896486;
   t1[19990] := 0.0789494;
   t1[19991] := 0.0681054;
   t1[19992] := 0.0571763;
   t1[19993] := 0.0462217;
   t1[19994] := 0.0353014;
   t1[19995] := 0.0244752;
   t1[19996] := 0.0138027;
   t1[19997] := 0.003338;
   t1[19998] := -0.0068928;
   t1[19999] := -0.0168727;
   t1[20000] := -0.0008921;
   t1[20001] := -0.0022787;
   t1[20002] := -0.0030907;
   t1[20003] := -0.0032964;
   t1[20004] := -0.0028641;
   t1[20005] := -0.0017621;
   t1[20006] := 4.14E-05;
   t1[20007] := 0.0025781;
   t1[20008] := 0.0058772;
   t1[20009] := 0.0099317;
   t1[20010] := 0.0147054;
   t1[20011] := 0.0201614;
   t1[20012] := 0.026263;
   t1[20013] := 0.0329734;
   t1[20014] := 0.0402556;
   t1[20015] := 0.0480728;
   t1[20016] := 0.0563883;
   t1[20017] := 0.0651652;
   t1[20018] := 0.0743666;
   t1[20019] := 0.0839557;
   t1[20020] := 0.0938957;
   t1[20021] := 0.1041497;
   t1[20022] := 0.114681;
   t1[20023] := 0.1254526;
   t1[20024] := 0.1364278;
   t1[20025] := 0.1475697;
   t1[20026] := 0.1588414;
   t1[20027] := 0.1702061;
   t1[20028] := 0.1816104;
   t1[20029] := 0.1929703;
   t1[20030] := 0.2041983;
   t1[20031] := 0.2152068;
   t1[20032] := 0.2259084;
   t1[20033] := 0.2362155;
   t1[20034] := 0.2460406;
   t1[20035] := 0.2552963;
   t1[20036] := 0.263895;
   t1[20037] := 0.2717492;
   t1[20038] := 0.2787713;
   t1[20039] := 0.284874;
   t1[20040] := 0.2899696;
   t1[20041] := 0.2939706;
   t1[20042] := 0.2967896;
   t1[20043] := 0.2983391;
   t1[20044] := 0.2985315;
   t1[20045] := 0.2972792;
   t1[20046] := 0.294495;
   t1[20047] := 0.2901186;
   t1[20048] := 0.2842278;
   t1[20049] := 0.2769434;
   t1[20050] := 0.1006214;
   t1[20051] := 0.0900307;
   t1[20052] := 0.0798032;
   t1[20053] := 0.0700324;
   t1[20054] := 0.0608116;
   t1[20055] := 0.0522343;
   t1[20056] := 0.0443938;
   t1[20057] := 0.0373836;
   t1[20058] := 0.0312934;
   t1[20059] := 0.0261583;
   t1[20060] := 0.0219696;
   t1[20061] := 0.018718;
   t1[20062] := 0.0163937;
   t1[20063] := 0.0149872;
   t1[20064] := 0.0144889;
   t1[20065] := 0.0148892;
   t1[20066] := 0.0161786;
   t1[20067] := 0.0183474;
   t1[20068] := 0.0213861;
   t1[20069] := 0.0252852;
   t1[20070] := 0.0300349;
   t1[20071] := 0.0356257;
   t1[20072] := 0.0420481;
   t1[20073] := 0.0492925;
   t1[20074] := 0.0573493;
   t1[20075] := 0.0662088;
   t1[20076] := 0.0758615;
   t1[20077] := 0.0862976;
   t1[20078] := 0.0974702;
   t1[20079] := 0.1092629;
   t1[20080] := 0.1215513;
   t1[20081] := 0.134211;
   t1[20082] := 0.1471177;
   t1[20083] := 0.1601472;
   t1[20084] := 0.1731751;
   t1[20085] := 0.186077;
   t1[20086] := 0.1987286;
   t1[20087] := 0.2110057;
   t1[20088] := 0.2227837;
   t1[20089] := 0.2339385;
   t1[20090] := 0.2443457;
   t1[20091] := 0.2538809;
   t1[20092] := 0.2624199;
   t1[20093] := 0.2698384;
   t1[20094] := 0.2760119;
   t1[20095] := 0.2808161;
   t1[20096] := 0.2841267;
   t1[20097] := 0.2858486;
   t1[20098] := 0.2860319;
   t1[20099] := 0.2847723;
   t1[20100] := 0.0050532;
   t1[20101] := 0.0067392;
   t1[20102] := 0.0082221;
   t1[20103] := 0.0094982;
   t1[20104] := 0.010564;
   t1[20105] := 0.0114159;
   t1[20106] := 0.0120503;
   t1[20107] := 0.0124636;
   t1[20108] := 0.0126532;
   t1[20109] := 0.012629;
   t1[20110] := 0.0124111;
   t1[20111] := 0.01202;
   t1[20112] := 0.0114758;
   t1[20113] := 0.0107991;
   t1[20114] := 0.0100102;
   t1[20115] := 0.0091295;
   t1[20116] := 0.0081773;
   t1[20117] := 0.007174;
   t1[20118] := 0.0061399;
   t1[20119] := 0.0050955;
   t1[20120] := 0.004061;
   t1[20121] := 0.003057;
   t1[20122] := 0.0021036;
   t1[20123] := 0.0012214;
   t1[20124] := 0.0004306;
   t1[20125] := -0.0002484;
   t1[20126] := -0.0007952;
   t1[20127] := -0.0011895;
   t1[20128] := -0.0014203;
   t1[20129] := -0.0014944;
   t1[20130] := -0.0014205;
   t1[20131] := -0.0012071;
   t1[20132] := -0.000863;
   t1[20133] := -0.0003969;
   t1[20134] := 0.0001826;
   t1[20135] := 0.0008668;
   t1[20136] := 0.0016471;
   t1[20137] := 0.0025147;
   t1[20138] := 0.003461;
   t1[20139] := 0.0044773;
   t1[20140] := 0.0055549;
   t1[20141] := 0.0066852;
   t1[20142] := 0.0078595;
   t1[20143] := 0.0090692;
   t1[20144] := 0.0103055;
   t1[20145] := 0.0115597;
   t1[20146] := 0.0128233;
   t1[20147] := 0.0140874;
   t1[20148] := 0.0153427;
   t1[20149] := 0.0165797;
   t1[20150] := 0.1193422;
   t1[20151] := 0.1142091;
   t1[20152] := 0.1093125;
   t1[20153] := 0.1046901;
   t1[20154] := 0.1003797;
   t1[20155] := 0.0964191;
   t1[20156] := 0.0928462;
   t1[20157] := 0.0896988;
   t1[20158] := 0.0870118;
   t1[20159] := 0.0847753;
   t1[20160] := 0.082944;
   t1[20161] := 0.0814718;
   t1[20162] := 0.0803124;
   t1[20163] := 0.0794197;
   t1[20164] := 0.0787474;
   t1[20165] := 0.0782495;
   t1[20166] := 0.0778797;
   t1[20167] := 0.0775919;
   t1[20168] := 0.0773397;
   t1[20169] := 0.0770772;
   t1[20170] := 0.076758;
   t1[20171] := 0.0763359;
   t1[20172] := 0.0757649;
   t1[20173] := 0.0749986;
   t1[20174] := 0.073991;
   t1[20175] := 0.0726958;
   t1[20176] := 0.0710669;
   t1[20177] := 0.0690583;
   t1[20178] := 0.0666513;
   t1[20179] := 0.0638794;
   t1[20180] := 0.0607816;
   t1[20181] := 0.057397;
   t1[20182] := 0.0537647;
   t1[20183] := 0.0499237;
   t1[20184] := 0.0459131;
   t1[20185] := 0.0417721;
   t1[20186] := 0.0375397;
   t1[20187] := 0.033255;
   t1[20188] := 0.028957;
   t1[20189] := 0.0246849;
   t1[20190] := 0.0204778;
   t1[20191] := 0.0163747;
   t1[20192] := 0.0124147;
   t1[20193] := 0.0086369;
   t1[20194] := 0.0050804;
   t1[20195] := 0.0017843;
   t1[20196] := -0.0012124;
   t1[20197] := -0.0038794;
   t1[20198] := -0.0062307;
   t1[20199] := -0.0082943;
   t1[20200] := 0.1559757;
   t1[20201] := 0.1469441;
   t1[20202] := 0.1379911;
   t1[20203] := 0.1291919;
   t1[20204] := 0.1206219;
   t1[20205] := 0.1123566;
   t1[20206] := 0.1044711;
   t1[20207] := 0.0970409;
   t1[20208] := 0.0901365;
   t1[20209] := 0.0837559;
   t1[20210] := 0.0778396;
   t1[20211] := 0.0723265;
   t1[20212] := 0.0671558;
   t1[20213] := 0.0622663;
   t1[20214] := 0.0575972;
   t1[20215] := 0.0530873;
   t1[20216] := 0.0486757;
   t1[20217] := 0.0443015;
   t1[20218] := 0.0399036;
   t1[20219] := 0.0354209;
   t1[20220] := 0.0307927;
   t1[20221] := 0.0259577;
   t1[20222] := 0.0208551;
   t1[20223] := 0.0154237;
   t1[20224] := 0.0096028;
   t1[20225] := 0.0033312;
   t1[20226] := -0.0034521;
   t1[20227] := -0.0108076;
   t1[20228] := -0.0187525;
   t1[20229] := -0.0272212;
   t1[20230] := -0.036139;
   t1[20231] := -0.0454311;
   t1[20232] := -0.055023;
   t1[20233] := -0.0648399;
   t1[20234] := -0.0748071;
   t1[20235] := -0.0848498;
   t1[20236] := -0.0948933;
   t1[20237] := -0.104863;
   t1[20238] := -0.1146841;
   t1[20239] := -0.124282;
   t1[20240] := -0.1335818;
   t1[20241] := -0.1425089;
   t1[20242] := -0.1509886;
   t1[20243] := -0.1589462;
   t1[20244] := -0.166307;
   t1[20245] := -0.1729962;
   t1[20246] := -0.1789391;
   t1[20247] := -0.1840752;
   t1[20248] := -0.1884141;
   t1[20249] := -0.1919876;
   t1[20250] := 0.0302589;
   t1[20251] := 0.0240423;
   t1[20252] := 0.0183947;
   t1[20253] := 0.0133858;
   t1[20254] := 0.0090853;
   t1[20255] := 0.0055629;
   t1[20256] := 0.0028882;
   t1[20257] := 0.001131;
   t1[20258] := 0.0003555;
   t1[20259] := 0.0005437;
   t1[20260] := 0.0016124;
   t1[20261] := 0.0034766;
   t1[20262] := 0.0060516;
   t1[20263] := 0.0092524;
   t1[20264] := 0.0129941;
   t1[20265] := 0.0171919;
   t1[20266] := 0.0217609;
   t1[20267] := 0.0266161;
   t1[20268] := 0.0316727;
   t1[20269] := 0.0368458;
   t1[20270] := 0.0420505;
   t1[20271] := 0.047202;
   t1[20272] := 0.0522153;
   t1[20273] := 0.0570055;
   t1[20274] := 0.0614878;
   t1[20275] := 0.0655773;
   t1[20276] := 0.0691891;
   t1[20277] := 0.0722386;
   t1[20278] := 0.0746798;
   t1[20279] := 0.0765393;
   t1[20280] := 0.0778522;
   t1[20281] := 0.0786532;
   t1[20282] := 0.0789773;
   t1[20283] := 0.0788594;
   t1[20284] := 0.0783344;
   t1[20285] := 0.0774371;
   t1[20286] := 0.0762025;
   t1[20287] := 0.0746655;
   t1[20288] := 0.0728609;
   t1[20289] := 0.0708236;
   t1[20290] := 0.0685886;
   t1[20291] := 0.0661907;
   t1[20292] := 0.0636648;
   t1[20293] := 0.0610459;
   t1[20294] := 0.0583688;
   t1[20295] := 0.0556683;
   t1[20296] := 0.0529795;
   t1[20297] := 0.0503326;
   t1[20298] := 0.0477351;
   t1[20299] := 0.0451873;
   t1[20300] := -0.0808457;
   t1[20301] := -0.0856393;
   t1[20302] := -0.0899749;
   t1[20303] := -0.0937563;
   t1[20304] := -0.0968873;
   t1[20305] := -0.0992716;
   t1[20306] := -0.1008129;
   t1[20307] := -0.101415;
   t1[20308] := -0.1009879;
   t1[20309] := -0.0995367;
   t1[20310] := -0.0971417;
   t1[20311] := -0.093885;
   t1[20312] := -0.0898488;
   t1[20313] := -0.0851153;
   t1[20314] := -0.0797668;
   t1[20315] := -0.0738855;
   t1[20316] := -0.0675535;
   t1[20317] := -0.0608531;
   t1[20318] := -0.0538665;
   t1[20319] := -0.0466759;
   t1[20320] := -0.0393634;
   t1[20321] := -0.0320114;
   t1[20322] := -0.024702;
   t1[20323] := -0.0175174;
   t1[20324] := -0.0105398;
   t1[20325] := -0.0038514;
   t1[20326] := 0.0024655;
   t1[20327] := 0.0083291;
   t1[20328] := 0.013699;
   t1[20329] := 0.0186131;
   t1[20330] := 0.0231181;
   t1[20331] := 0.0272606;
   t1[20332] := 0.0310875;
   t1[20333] := 0.0346453;
   t1[20334] := 0.0379809;
   t1[20335] := 0.0411408;
   t1[20336] := 0.0441719;
   t1[20337] := 0.0471207;
   t1[20338] := 0.0500341;
   t1[20339] := 0.0529586;
   t1[20340] := 0.0559411;
   t1[20341] := 0.0590281;
   t1[20342] := 0.0622665;
   t1[20343] := 0.0657028;
   t1[20344] := 0.0693839;
   t1[20345] := 0.0733563;
   t1[20346] := 0.0776669;
   t1[20347] := 0.082347;
   t1[20348] := 0.0873516;
   t1[20349] := 0.0926117;
   t1[20350] := 0.2293762;
   t1[20351] := 0.2240999;
   t1[20352] := 0.2184374;
   t1[20353] := 0.2123844;
   t1[20354] := 0.2059362;
   t1[20355] := 0.1990884;
   t1[20356] := 0.1918364;
   t1[20357] := 0.1841759;
   t1[20358] := 0.1761033;
   t1[20359] := 0.1676282;
   t1[20360] := 0.1587709;
   t1[20361] := 0.1495522;
   t1[20362] := 0.1399926;
   t1[20363] := 0.1301127;
   t1[20364] := 0.1199331;
   t1[20365] := 0.1094744;
   t1[20366] := 0.0987572;
   t1[20367] := 0.0878021;
   t1[20368] := 0.0766298;
   t1[20369] := 0.0652608;
   t1[20370] := 0.0537157;
   t1[20371] := 0.0420152;
   t1[20372] := 0.0301798;
   t1[20373] := 0.0182302;
   t1[20374] := 0.0061868;
   t1[20375] := -0.0059295;
   t1[20376] := -0.0180983;
   t1[20377] := -0.0302989;
   t1[20378] := -0.0425065;
   t1[20379] := -0.0546886;
   t1[20380] := -0.0668115;
   t1[20381] := -0.0788417;
   t1[20382] := -0.0907459;
   t1[20383] := -0.1024903;
   t1[20384] := -0.1140417;
   t1[20385] := -0.1253664;
   t1[20386] := -0.1364309;
   t1[20387] := -0.1472017;
   t1[20388] := -0.1576453;
   t1[20389] := -0.1677282;
   t1[20390] := -0.177417;
   t1[20391] := -0.1866779;
   t1[20392] := -0.1954777;
   t1[20393] := -0.2037828;
   t1[20394] := -0.2115596;
   t1[20395] := -0.2187747;
   t1[20396] := -0.2253944;
   t1[20397] := -0.2313912;
   t1[20398] := -0.2367659;
   t1[20399] := -0.2415285;
   t1[20400] := -0.0665781;
   t1[20401] := -0.0756864;
   t1[20402] := -0.0840258;
   t1[20403] := -0.0914937;
   t1[20404] := -0.0979875;
   t1[20405] := -0.1034044;
   t1[20406] := -0.1076418;
   t1[20407] := -0.110597;
   t1[20408] := -0.1121747;
   t1[20409] := -0.11239;
   t1[20410] := -0.1113457;
   t1[20411] := -0.1091466;
   t1[20412] := -0.1058976;
   t1[20413] := -0.1017037;
   t1[20414] := -0.0966698;
   t1[20415] := -0.0909009;
   t1[20416] := -0.0845018;
   t1[20417] := -0.0775775;
   t1[20418] := -0.070233;
   t1[20419] := -0.0625731;
   t1[20420] := -0.0547028;
   t1[20421] := -0.046727;
   t1[20422] := -0.0387506;
   t1[20423] := -0.0308786;
   t1[20424] := -0.023216;
   t1[20425] := -0.0158675;
   t1[20426] := -0.0089383;
   t1[20427] := -0.0025327;
   t1[20428] := 0.0032941;
   t1[20429] := 0.0085803;
   t1[20430] := 0.0133748;
   t1[20431] := 0.0177263;
   t1[20432] := 0.0216834;
   t1[20433] := 0.025295;
   t1[20434] := 0.0286098;
   t1[20435] := 0.0316765;
   t1[20436] := 0.0345439;
   t1[20437] := 0.0372607;
   t1[20438] := 0.0398757;
   t1[20439] := 0.0424376;
   t1[20440] := 0.0449952;
   t1[20441] := 0.0475971;
   t1[20442] := 0.0502922;
   t1[20443] := 0.0531292;
   t1[20444] := 0.0561569;
   t1[20445] := 0.0594239;
   t1[20446] := 0.062979;
   t1[20447] := 0.0668552;
   t1[20448] := 0.0710065;
   t1[20449] := 0.0753623;
   t1[20450] := -0.2079995;
   t1[20451] := -0.214729;
   t1[20452] := -0.2210183;
   t1[20453] := -0.22675;
   t1[20454] := -0.2318069;
   t1[20455] := -0.2360717;
   t1[20456] := -0.2394271;
   t1[20457] := -0.2417559;
   t1[20458] := -0.2429459;
   t1[20459] := -0.2429626;
   t1[20460] := -0.2418332;
   t1[20461] := -0.239586;
   t1[20462] := -0.2362499;
   t1[20463] := -0.2318534;
   t1[20464] := -0.226425;
   t1[20465] := -0.2199935;
   t1[20466] := -0.2125875;
   t1[20467] := -0.2042355;
   t1[20468] := -0.1949662;
   t1[20469] := -0.1848082;
   t1[20470] := -0.1737901;
   t1[20471] := -0.1619405;
   t1[20472] := -0.1492881;
   t1[20473] := -0.1358614;
   t1[20474] := -0.1216891;
   t1[20475] := -0.1067998;
   t1[20476] := -0.0912221;
   t1[20477] := -0.0749847;
   t1[20478] := -0.0581369;
   t1[20479] := -0.0407662;
   t1[20480] := -0.0229645;
   t1[20481] := -0.0048236;
   t1[20482] := 0.0135645;
   t1[20483] := 0.0321079;
   t1[20484] := 0.0507148;
   t1[20485] := 0.0692932;
   t1[20486] := 0.0877513;
   t1[20487] := 0.1059972;
   t1[20488] := 0.123939;
   t1[20489] := 0.1414848;
   t1[20490] := 0.1585426;
   t1[20491] := 0.1750207;
   t1[20492] := 0.190827;
   t1[20493] := 0.2058699;
   t1[20494] := 0.2200573;
   t1[20495] := 0.2332973;
   t1[20496] := 0.245498;
   t1[20497] := 0.2565814;
   t1[20498] := 0.2665374;
   t1[20499] := 0.2753775;
   t1[20500] := 0.1881377;
   t1[20501] := 0.1915277;
   t1[20502] := 0.1939553;
   t1[20503] := 0.1952612;
   t1[20504] := 0.1952864;
   t1[20505] := 0.1938717;
   t1[20506] := 0.1908578;
   t1[20507] := 0.1860857;
   t1[20508] := 0.1794081;
   t1[20509] := 0.1708636;
   t1[20510] := 0.1606369;
   t1[20511] := 0.1489166;
   t1[20512] := 0.1358914;
   t1[20513] := 0.1217499;
   t1[20514] := 0.1066808;
   t1[20515] := 0.0908728;
   t1[20516] := 0.0745145;
   t1[20517] := 0.0577945;
   t1[20518] := 0.0409016;
   t1[20519] := 0.0240243;
   t1[20520] := 0.0073514;
   t1[20521] := -0.0089286;
   t1[20522] := -0.0246269;
   t1[20523] := -0.039555;
   t1[20524] := -0.0535241;
   t1[20525] := -0.0663456;
   t1[20526] := -0.0778308;
   t1[20527] := -0.087792;
   t1[20528] := -0.0961361;
   t1[20529] := -0.1029493;
   t1[20530] := -0.1083381;
   t1[20531] := -0.1124091;
   t1[20532] := -0.1152685;
   t1[20533] := -0.1170228;
   t1[20534] := -0.1177784;
   t1[20535] := -0.1176418;
   t1[20536] := -0.1167194;
   t1[20537] := -0.1151175;
   t1[20538] := -0.1129428;
   t1[20539] := -0.1103014;
   t1[20540] := -0.1073;
   t1[20541] := -0.1040449;
   t1[20542] := -0.1006425;
   t1[20543] := -0.0971993;
   t1[20544] := -0.0938217;
   t1[20545] := -0.090616;
   t1[20546] := -0.0876889;
   t1[20547] := -0.0851268;
   t1[20548] := -0.0829181;
   t1[20549] := -0.08102;
   t1[20550] := 0.3099137;
   t1[20551] := 0.3104934;
   t1[20552] := 0.3104255;
   t1[20553] := 0.3096267;
   t1[20554] := 0.3080136;
   t1[20555] := 0.3055028;
   t1[20556] := 0.3020107;
   t1[20557] := 0.2974539;
   t1[20558] := 0.291755;
   t1[20559] := 0.2849257;
   t1[20560] := 0.2770485;
   t1[20561] := 0.268208;
   t1[20562] := 0.2584884;
   t1[20563] := 0.2479741;
   t1[20564] := 0.2367496;
   t1[20565] := 0.2248992;
   t1[20566] := 0.2125074;
   t1[20567] := 0.1996585;
   t1[20568] := 0.1864369;
   t1[20569] := 0.172927;
   t1[20570] := 0.1592133;
   t1[20571] := 0.14538;
   t1[20572] := 0.1315116;
   t1[20573] := 0.1176925;
   t1[20574] := 0.1040071;
   t1[20575] := 0.0905397;
   t1[20576] := 0.0773749;
   t1[20577] := 0.0645965;
   t1[20578] := 0.0522519;
   t1[20579] := 0.0403183;
   t1[20580] := 0.0287653;
   t1[20581] := 0.0175623;
   t1[20582] := 0.006679;
   t1[20583] := -0.0039153;
   t1[20584] := -0.0142509;
   t1[20585] := -0.0243583;
   t1[20586] := -0.0342682;
   t1[20587] := -0.0440108;
   t1[20588] := -0.0536167;
   t1[20589] := -0.0631165;
   t1[20590] := -0.0725405;
   t1[20591] := -0.0819192;
   t1[20592] := -0.0912833;
   t1[20593] := -0.100663;
   t1[20594] := -0.110089;
   t1[20595] := -0.1195917;
   t1[20596] := -0.1292015;
   t1[20597] := -0.1389386;
   t1[20598] := -0.148771;
   t1[20599] := -0.1586504;
   t1[20600] := -0.1184668;
   t1[20601] := -0.1136256;
   t1[20602] := -0.1086983;
   t1[20603] := -0.1036999;
   t1[20604] := -0.0986453;
   t1[20605] := -0.0935495;
   t1[20606] := -0.0884274;
   t1[20607] := -0.0832939;
   t1[20608] := -0.0781617;
   t1[20609] := -0.0730062;
   t1[20610] := -0.0677739;
   t1[20611] := -0.0624104;
   t1[20612] := -0.0568614;
   t1[20613] := -0.0510724;
   t1[20614] := -0.0449892;
   t1[20615] := -0.0385572;
   t1[20616] := -0.0317222;
   t1[20617] := -0.0244298;
   t1[20618] := -0.0166256;
   t1[20619] := -0.0082553;
   t1[20620] := 0.0007356;
   t1[20621] := 0.0104014;
   t1[20622] := 0.0207964;
   t1[20623] := 0.0319752;
   t1[20624] := 0.0439919;
   t1[20625] := 0.056901;
   t1[20626] := 0.0707569;
   t1[20627] := 0.0856132;
   t1[20628] := 0.1014512;
   t1[20629] := 0.1181145;
   t1[20630] := 0.1354313;
   t1[20631] := 0.1532297;
   t1[20632] := 0.1713383;
   t1[20633] := 0.189585;
   t1[20634] := 0.2077983;
   t1[20635] := 0.2258063;
   t1[20636] := 0.2434374;
   t1[20637] := 0.2605197;
   t1[20638] := 0.2768814;
   t1[20639] := 0.2923509;
   t1[20640] := 0.3067565;
   t1[20641] := 0.3199262;
   t1[20642] := 0.3316885;
   t1[20643] := 0.3418716;
   t1[20644] := 0.3503036;
   t1[20645] := 0.3568129;
   t1[20646] := 0.3612277;
   t1[20647] := 0.3634188;
   t1[20648] := 0.3634697;
   t1[20649] := 0.3615301;
   t1[20650] := -0.091948;
   t1[20651] := -0.0946389;
   t1[20652] := -0.0967835;
   t1[20653] := -0.0983482;
   t1[20654] := -0.0992989;
   t1[20655] := -0.0996019;
   t1[20656] := -0.0992233;
   t1[20657] := -0.0981292;
   t1[20658] := -0.0962892;
   t1[20659] := -0.0937279;
   t1[20660] := -0.0905124;
   t1[20661] := -0.0867115;
   t1[20662] := -0.0823936;
   t1[20663] := -0.0776273;
   t1[20664] := -0.0724812;
   t1[20665] := -0.0670238;
   t1[20666] := -0.0613236;
   t1[20667] := -0.0554493;
   t1[20668] := -0.0494693;
   t1[20669] := -0.0434523;
   t1[20670] := -0.0374667;
   t1[20671] := -0.0315812;
   t1[20672] := -0.0258643;
   t1[20673] := -0.0203845;
   t1[20674] := -0.0152104;
   t1[20675] := -0.0104106;
   t1[20676] := -0.0060536;
   t1[20677] := -0.0022076;
   t1[20678] := 0.0011018;
   t1[20679] := 0.0039296;
   t1[20680] := 0.0063398;
   t1[20681] := 0.0083963;
   t1[20682] := 0.0101633;
   t1[20683] := 0.0117047;
   t1[20684] := 0.0130845;
   t1[20685] := 0.0143668;
   t1[20686] := 0.0156154;
   t1[20687] := 0.0168946;
   t1[20688] := 0.0182681;
   t1[20689] := 0.0198002;
   t1[20690] := 0.0215547;
   t1[20691] := 0.0235956;
   t1[20692] := 0.0259871;
   t1[20693] := 0.028793;
   t1[20694] := 0.0320775;
   t1[20695] := 0.0359044;
   t1[20696] := 0.0403379;
   t1[20697] := 0.0454208;
   t1[20698] := 0.0510906;
   t1[20699] := 0.0572519;
   t1[20700] := -0.0519979;
   t1[20701] := -0.0398461;
   t1[20702] := -0.0280016;
   t1[20703] := -0.0165445;
   t1[20704] := -0.0055546;
   t1[20705] := 0.0048879;
   t1[20706] := 0.0147033;
   t1[20707] := 0.0238115;
   t1[20708] := 0.0321374;
   t1[20709] := 0.0396818;
   t1[20710] := 0.0465054;
   t1[20711] := 0.0526702;
   t1[20712] := 0.0582385;
   t1[20713] := 0.0632722;
   t1[20714] := 0.0678337;
   t1[20715] := 0.071985;
   t1[20716] := 0.0757883;
   t1[20717] := 0.0793058;
   t1[20718] := 0.0825995;
   t1[20719] := 0.0857317;
   t1[20720] := 0.0887645;
   t1[20721] := 0.09176;
   t1[20722] := 0.0947804;
   t1[20723] := 0.0978879;
   t1[20724] := 0.1011445;
   t1[20725] := 0.1046124;
   t1[20726] := 0.1083539;
   t1[20727] := 0.1124306;
   t1[20728] := 0.1168682;
   t1[20729] := 0.1216235;
   t1[20730] := 0.1266455;
   t1[20731] := 0.1318834;
   t1[20732] := 0.1372863;
   t1[20733] := 0.1428033;
   t1[20734] := 0.1483834;
   t1[20735] := 0.1539759;
   t1[20736] := 0.1595298;
   t1[20737] := 0.1649943;
   t1[20738] := 0.1703183;
   t1[20739] := 0.1754512;
   t1[20740] := 0.1803419;
   t1[20741] := 0.1849396;
   t1[20742] := 0.1891934;
   t1[20743] := 0.1930524;
   t1[20744] := 0.1964656;
   t1[20745] := 0.1993823;
   t1[20746] := 0.2017516;
   t1[20747] := 0.2035316;
   t1[20748] := 0.2047262;
   t1[20749] := 0.2053535;
   t1[20750] := 0.0139801;
   t1[20751] := 0.0327884;
   t1[20752] := 0.0509511;
   t1[20753] := 0.0682511;
   t1[20754] := 0.0844717;
   t1[20755] := 0.0993961;
   t1[20756] := 0.1128075;
   t1[20757] := 0.124489;
   t1[20758] := 0.1342357;
   t1[20759] := 0.1420261;
   t1[20760] := 0.1479834;
   t1[20761] := 0.1522347;
   t1[20762] := 0.1549069;
   t1[20763] := 0.1561271;
   t1[20764] := 0.1560223;
   t1[20765] := 0.1547194;
   t1[20766] := 0.1523457;
   t1[20767] := 0.1490279;
   t1[20768] := 0.1448933;
   t1[20769] := 0.1400687;
   t1[20770] := 0.1346813;
   t1[20771] := 0.128858;
   t1[20772] := 0.1227258;
   t1[20773] := 0.1164118;
   t1[20774] := 0.1100431;
   t1[20775] := 0.1037465;
   t1[20776] := 0.0976492;
   t1[20777] := 0.0918778;
   t1[20778] := 0.0865192;
   t1[20779] := 0.0815844;
   t1[20780] := 0.0770762;
   t1[20781] := 0.0729975;
   t1[20782] := 0.069351;
   t1[20783] := 0.0661394;
   t1[20784] := 0.0633654;
   t1[20785] := 0.0610319;
   t1[20786] := 0.0591416;
   t1[20787] := 0.0576973;
   t1[20788] := 0.0567017;
   t1[20789] := 0.0561575;
   t1[20790] := 0.0560676;
   t1[20791] := 0.0564346;
   t1[20792] := 0.0572614;
   t1[20793] := 0.0585508;
   t1[20794] := 0.0603053;
   t1[20795] := 0.0625279;
   t1[20796] := 0.0652213;
   t1[20797] := 0.0683785;
   t1[20798] := 0.0719446;
   t1[20799] := 0.0758494;
   t1[20800] := -0.0209548;
   t1[20801] := -0.0203117;
   t1[20802] := -0.0194967;
   t1[20803] := -0.0185084;
   t1[20804] := -0.0173451;
   t1[20805] := -0.0160056;
   t1[20806] := -0.0144882;
   t1[20807] := -0.0127916;
   t1[20808] := -0.0109143;
   t1[20809] := -0.0088567;
   t1[20810] := -0.0066203;
   t1[20811] := -0.0042068;
   t1[20812] := -0.0016177;
   t1[20813] := 0.0011453;
   t1[20814] := 0.0040806;
   t1[20815] := 0.0071865;
   t1[20816] := 0.0104616;
   t1[20817] := 0.0139041;
   t1[20818] := 0.0175125;
   t1[20819] := 0.0212851;
   t1[20820] := 0.0252203;
   t1[20821] := 0.0293165;
   t1[20822] := 0.0335721;
   t1[20823] := 0.0379855;
   t1[20824] := 0.042555;
   t1[20825] := 0.047279;
   t1[20826] := 0.052156;
   t1[20827] := 0.0571842;
   t1[20828] := 0.0623495;
   t1[20829] := 0.0676145;
   t1[20830] := 0.072939;
   t1[20831] := 0.078283;
   t1[20832] := 0.0836064;
   t1[20833] := 0.088869;
   t1[20834] := 0.0940309;
   t1[20835] := 0.0990518;
   t1[20836] := 0.1038918;
   t1[20837] := 0.1085107;
   t1[20838] := 0.1128684;
   t1[20839] := 0.1169249;
   t1[20840] := 0.12064;
   t1[20841] := 0.1239737;
   t1[20842] := 0.1268858;
   t1[20843] := 0.1293363;
   t1[20844] := 0.1312851;
   t1[20845] := 0.1326921;
   t1[20846] := 0.1335172;
   t1[20847] := 0.133731;
   t1[20848] := 0.133357;
   t1[20849] := 0.1324356;
   t1[20850] := -0.1402293;
   t1[20851] := -0.1278123;
   t1[20852] := -0.1153219;
   t1[20853] := -0.1028302;
   t1[20854] := -0.0904093;
   t1[20855] := -0.0781312;
   t1[20856] := -0.0660679;
   t1[20857] := -0.0542916;
   t1[20858] := -0.0428716;
   t1[20859] := -0.0318349;
   t1[20860] := -0.0211754;
   t1[20861] := -0.0108859;
   t1[20862] := -0.0009594;
   t1[20863] := 0.0086114;
   t1[20864] := 0.0178334;
   t1[20865] := 0.0267139;
   t1[20866] := 0.0352599;
   t1[20867] := 0.0434785;
   t1[20868] := 0.0513768;
   t1[20869] := 0.058962;
   t1[20870] := 0.0662411;
   t1[20871] := 0.0732214;
   t1[20872] := 0.0799097;
   t1[20873] := 0.0863134;
   t1[20874] := 0.0924395;
   t1[20875] := 0.0982951;
   t1[20876] := 0.1038873;
   t1[20877] := 0.1092232;
   t1[20878] := 0.1143034;
   t1[20879] := 0.1191161;
   t1[20880] := 0.1236483;
   t1[20881] := 0.127887;
   t1[20882] := 0.131819;
   t1[20883] := 0.1354314;
   t1[20884] := 0.1387111;
   t1[20885] := 0.1416449;
   t1[20886] := 0.1442199;
   t1[20887] := 0.146423;
   t1[20888] := 0.1482412;
   t1[20889] := 0.1496613;
   t1[20890] := 0.1506703;
   t1[20891] := 0.1512552;
   t1[20892] := 0.1514029;
   t1[20893] := 0.1511003;
   t1[20894] := 0.1503344;
   t1[20895] := 0.1490922;
   t1[20896] := 0.1473604;
   t1[20897] := 0.145133;
   t1[20898] := 0.142437;
   t1[20899] := 0.1393104;
   t1[20900] := -0.0203112;
   t1[20901] := -0.0134685;
   t1[20902] := -0.0065542;
   t1[20903] := 0.0003836;
   t1[20904] := 0.0072966;
   t1[20905] := 0.0141366;
   t1[20906] := 0.0208553;
   t1[20907] := 0.0274046;
   t1[20908] := 0.0337381;
   t1[20909] := 0.039841;
   t1[20910] := 0.0457231;
   t1[20911] := 0.0513949;
   t1[20912] := 0.0568668;
   t1[20913] := 0.0621493;
   t1[20914] := 0.0672529;
   t1[20915] := 0.072188;
   t1[20916] := 0.0769651;
   t1[20917] := 0.0815946;
   t1[20918] := 0.086087;
   t1[20919] := 0.0904529;
   t1[20920] := 0.0947025;
   t1[20921] := 0.0988465;
   t1[20922] := 0.1028953;
   t1[20923] := 0.1068593;
   t1[20924] := 0.1107489;
   t1[20925] := 0.1145748;
   t1[20926] := 0.1183473;
   t1[20927] := 0.1220767;
   t1[20928] := 0.1257661;
   t1[20929] := 0.1294038;
   t1[20930] := 0.1329767;
   t1[20931] := 0.1364716;
   t1[20932] := 0.1398756;
   t1[20933] := 0.1431753;
   t1[20934] := 0.1463578;
   t1[20935] := 0.1494099;
   t1[20936] := 0.1523185;
   t1[20937] := 0.1550704;
   t1[20938] := 0.1576525;
   t1[20939] := 0.1600517;
   t1[20940] := 0.162255;
   t1[20941] := 0.164249;
   t1[20942] := 0.1660208;
   t1[20943] := 0.1675572;
   t1[20944] := 0.1688451;
   t1[20945] := 0.1698714;
   t1[20946] := 0.1706229;
   t1[20947] := 0.1710883;
   t1[20948] := 0.1712647;
   t1[20949] := 0.171152;
   t1[20950] := 0.046874;
   t1[20951] := 0.0361466;
   t1[20952] := 0.0258332;
   t1[20953] := 0.0159921;
   t1[20954] := 0.0066817;
   t1[20955] := -0.0020396;
   t1[20956] := -0.0101134;
   t1[20957] := -0.0174814;
   t1[20958] := -0.024087;
   t1[20959] := -0.0299034;
   t1[20960] := -0.0349269;
   t1[20961] := -0.0391544;
   t1[20962] := -0.0425831;
   t1[20963] := -0.0452097;
   t1[20964] := -0.0470314;
   t1[20965] := -0.0480451;
   t1[20966] := -0.0482477;
   t1[20967] := -0.0476362;
   t1[20968] := -0.0462077;
   t1[20969] := -0.043959;
   t1[20970] := -0.0408872;
   t1[20971] := -0.0369892;
   t1[20972] := -0.032262;
   t1[20973] := -0.0267026;
   t1[20974] := -0.0203079;
   t1[20975] := -0.013075;
   t1[20976] := -0.0050008;
   t1[20977] := 0.0039174;
   t1[20978] := 0.0136476;
   t1[20979] := 0.024092;
   t1[20980] := 0.0351453;
   t1[20981] := 0.0467023;
   t1[20982] := 0.0586579;
   t1[20983] := 0.0709068;
   t1[20984] := 0.0833438;
   t1[20985] := 0.0958637;
   t1[20986] := 0.1083613;
   t1[20987] := 0.1207315;
   t1[20988] := 0.1328689;
   t1[20989] := 0.1446684;
   t1[20990] := 0.1560249;
   t1[20991] := 0.1668329;
   t1[20992] := 0.1769875;
   t1[20993] := 0.1863834;
   t1[20994] := 0.1949153;
   t1[20995] := 0.2024781;
   t1[20996] := 0.2089665;
   t1[20997] := 0.2142964;
   t1[20998] := 0.218488;
   t1[20999] := 0.2215942;
   t1[21000] := -0.0061098;
   t1[21001] := -0.009897;
   t1[21002] := -0.0139381;
   t1[21003] := -0.0182364;
   t1[21004] := -0.0227955;
   t1[21005] := -0.0276188;
   t1[21006] := -0.0327098;
   t1[21007] := -0.0380719;
   t1[21008] := -0.0437061;
   t1[21009] := -0.0495736;
   t1[21010] := -0.0556047;
   t1[21011] := -0.0617285;
   t1[21012] := -0.0678745;
   t1[21013] := -0.0739718;
   t1[21014] := -0.0799497;
   t1[21015] := -0.0857377;
   t1[21016] := -0.0912649;
   t1[21017] := -0.0964606;
   t1[21018] := -0.1012542;
   t1[21019] := -0.1055749;
   t1[21020] := -0.1093521;
   t1[21021] := -0.1125149;
   t1[21022] := -0.1149928;
   t1[21023] := -0.116715;
   t1[21024] := -0.1176107;
   t1[21025] := -0.1176094;
   t1[21026] := -0.1166402;
   t1[21027] := -0.1146329;
   t1[21028] := -0.1115672;
   t1[21029] := -0.1075169;
   t1[21030] := -0.1025666;
   t1[21031] := -0.0968008;
   t1[21032] := -0.0903041;
   t1[21033] := -0.0831611;
   t1[21034] := -0.0754562;
   t1[21035] := -0.0672741;
   t1[21036] := -0.0586992;
   t1[21037] := -0.049816;
   t1[21038] := -0.0407093;
   t1[21039] := -0.0314633;
   t1[21040] := -0.0221628;
   t1[21041] := -0.0128923;
   t1[21042] := -0.0037362;
   t1[21043] := 0.0052209;
   t1[21044] := 0.0138944;
   t1[21045] := 0.0221997;
   t1[21046] := 0.0300524;
   t1[21047] := 0.0373809;
   t1[21048] := 0.0441785;
   t1[21049] := 0.0504587;
   t1[21050] := 0.0525412;
   t1[21051] := 0.0511629;
   t1[21052] := 0.0500092;
   t1[21053] := 0.049101;
   t1[21054] := 0.0484592;
   t1[21055] := 0.0481049;
   t1[21056] := 0.0480589;
   t1[21057] := 0.0483423;
   t1[21058] := 0.0489746;
   t1[21059] := 0.049954;
   t1[21060] := 0.0512616;
   t1[21061] := 0.0528784;
   t1[21062] := 0.0547849;
   t1[21063] := 0.0569622;
   t1[21064] := 0.0593908;
   t1[21065] := 0.0620516;
   t1[21066] := 0.0649253;
   t1[21067] := 0.0679928;
   t1[21068] := 0.0712348;
   t1[21069] := 0.0746321;
   t1[21070] := 0.0781655;
   t1[21071] := 0.0818158;
   t1[21072] := 0.0855636;
   t1[21073] := 0.0893899;
   t1[21074] := 0.0932754;
   t1[21075] := 0.0972008;
   t1[21076] := 0.101147;
   t1[21077] := 0.1050947;
   t1[21078] := 0.109027;
   t1[21079] := 0.1129312;
   t1[21080] := 0.1167952;
   t1[21081] := 0.1206066;
   t1[21082] := 0.1243533;
   t1[21083] := 0.1280232;
   t1[21084] := 0.1316039;
   t1[21085] := 0.1350833;
   t1[21086] := 0.1384492;
   t1[21087] := 0.1416894;
   t1[21088] := 0.1447917;
   t1[21089] := 0.1477438;
   t1[21090] := 0.1505336;
   t1[21091] := 0.1531489;
   t1[21092] := 0.1555775;
   t1[21093] := 0.1578071;
   t1[21094] := 0.1598255;
   t1[21095] := 0.1616207;
   t1[21096] := 0.1631802;
   t1[21097] := 0.164495;
   t1[21098] := 0.1655703;
   t1[21099] := 0.1664159;
   t1[21100] := 0.0825259;
   t1[21101] := 0.0878747;
   t1[21102] := 0.092803;
   t1[21103] := 0.09725;
   t1[21104] := 0.1011553;
   t1[21105] := 0.1044581;
   t1[21106] := 0.1070977;
   t1[21107] := 0.1090136;
   t1[21108] := 0.1101494;
   t1[21109] := 0.1105138;
   t1[21110] := 0.1101673;
   t1[21111] := 0.1091714;
   t1[21112] := 0.107588;
   t1[21113] := 0.1054786;
   t1[21114] := 0.1029049;
   t1[21115] := 0.0999287;
   t1[21116] := 0.0966116;
   t1[21117] := 0.0930154;
   t1[21118] := 0.0892016;
   t1[21119] := 0.085232;
   t1[21120] := 0.0811683;
   t1[21121] := 0.0770722;
   t1[21122] := 0.0730053;
   t1[21123] := 0.0690294;
   t1[21124] := 0.065206;
   t1[21125] := 0.061597;
   t1[21126] := 0.058264;
   t1[21127] := 0.0552684;
   t1[21128] := 0.0526507;
   t1[21129] := 0.050411;
   t1[21130] := 0.048545;
   t1[21131] := 0.0470485;
   t1[21132] := 0.0459171;
   t1[21133] := 0.0451466;
   t1[21134] := 0.0447326;
   t1[21135] := 0.0446709;
   t1[21136] := 0.0449572;
   t1[21137] := 0.0455872;
   t1[21138] := 0.0465567;
   t1[21139] := 0.0478613;
   t1[21140] := 0.0494967;
   t1[21141] := 0.0514586;
   t1[21142] := 0.0537429;
   t1[21143] := 0.0563451;
   t1[21144] := 0.059261;
   t1[21145] := 0.0624863;
   t1[21146] := 0.0660167;
   t1[21147] := 0.069843;
   t1[21148] := 0.0739313;
   t1[21149] := 0.0782398;
   t1[21150] := 0.1141067;
   t1[21151] := 0.1097303;
   t1[21152] := 0.105666;
   t1[21153] := 0.1019882;
   t1[21154] := 0.0987717;
   t1[21155] := 0.0960911;
   t1[21156] := 0.0940209;
   t1[21157] := 0.092636;
   t1[21158] := 0.0920057;
   t1[21159] := 0.0921193;
   t1[21160] := 0.0929031;
   t1[21161] := 0.0942816;
   t1[21162] := 0.0961793;
   t1[21163] := 0.0985207;
   t1[21164] := 0.1012303;
   t1[21165] := 0.1042327;
   t1[21166] := 0.1074525;
   t1[21167] := 0.110814;
   t1[21168] := 0.1142418;
   t1[21169] := 0.1176605;
   t1[21170] := 0.1209946;
   t1[21171] := 0.1241685;
   t1[21172] := 0.1271069;
   t1[21173] := 0.1297342;
   t1[21174] := 0.131975;
   t1[21175] := 0.1337537;
   t1[21176] := 0.134995;
   t1[21177] := 0.1356235;
   t1[21178] := 0.1355985;
   t1[21179] := 0.1349439;
   t1[21180] := 0.1336911;
   t1[21181] := 0.1318713;
   t1[21182] := 0.1295159;
   t1[21183] := 0.126656;
   t1[21184] := 0.1233231;
   t1[21185] := 0.1195484;
   t1[21186] := 0.1153632;
   t1[21187] := 0.1107988;
   t1[21188] := 0.1058864;
   t1[21189] := 0.1006574;
   t1[21190] := 0.0951432;
   t1[21191] := 0.0893748;
   t1[21192] := 0.0833837;
   t1[21193] := 0.0772012;
   t1[21194] := 0.0708585;
   t1[21195] := 0.0643869;
   t1[21196] := 0.0578178;
   t1[21197] := 0.0511814;
   t1[21198] := 0.0445032;
   t1[21199] := 0.0378071;
   t1[21200] := -0.0047682;
   t1[21201] := 0.0052685;
   t1[21202] := 0.0152905;
   t1[21203] := 0.0251887;
   t1[21204] := 0.034854;
   t1[21205] := 0.0441773;
   t1[21206] := 0.0530495;
   t1[21207] := 0.0613615;
   t1[21208] := 0.0690082;
   t1[21209] := 0.0759458;
   t1[21210] := 0.0821789;
   t1[21211] := 0.0877134;
   t1[21212] := 0.0925552;
   t1[21213] := 0.0967101;
   t1[21214] := 0.1001842;
   t1[21215] := 0.1029832;
   t1[21216] := 0.105113;
   t1[21217] := 0.1065796;
   t1[21218] := 0.1073888;
   t1[21219] := 0.1075466;
   t1[21220] := 0.1070588;
   t1[21221] := 0.1059313;
   t1[21222] := 0.10417;
   t1[21223] := 0.1017808;
   t1[21224] := 0.0987696;
   t1[21225] := 0.0951422;
   t1[21226] := 0.0909047;
   t1[21227] := 0.0860631;
   t1[21228] := 0.0806607;
   t1[21229] := 0.0748109;
   t1[21230] := 0.0686348;
   t1[21231] := 0.0622536;
   t1[21232] := 0.0557884;
   t1[21233] := 0.0493605;
   t1[21234] := 0.0430909;
   t1[21235] := 0.0371009;
   t1[21236] := 0.0315116;
   t1[21237] := 0.0264442;
   t1[21238] := 0.0220198;
   t1[21239] := 0.0183597;
   t1[21240] := 0.015585;
   t1[21241] := 0.0138168;
   t1[21242] := 0.0131764;
   t1[21243] := 0.0137848;
   t1[21244] := 0.0157633;
   t1[21245] := 0.0192331;
   t1[21246] := 0.0243153;
   t1[21247] := 0.0310951;
   t1[21248] := 0.0394778;
   t1[21249] := 0.0493127;
   t1[21250] := -0.0994751;
   t1[21251] := -0.0964376;
   t1[21252] := -0.0930327;
   t1[21253] := -0.0892771;
   t1[21254] := -0.0851872;
   t1[21255] := -0.0807795;
   t1[21256] := -0.0760706;
   t1[21257] := -0.0710769;
   t1[21258] := -0.0658163;
   t1[21259] := -0.0603274;
   t1[21260] := -0.0546647;
   t1[21261] := -0.0488836;
   t1[21262] := -0.0430391;
   t1[21263] := -0.0371865;
   t1[21264] := -0.031381;
   t1[21265] := -0.0256776;
   t1[21266] := -0.0201316;
   t1[21267] := -0.0147983;
   t1[21268] := -0.0097326;
   t1[21269] := -0.0049899;
   t1[21270] := -0.0006252;
   t1[21271] := 0.0033061;
   t1[21272] := 0.0067491;
   t1[21273] := 0.0096484;
   t1[21274] := 0.0119489;
   t1[21275] := 0.0135954;
   t1[21276] := 0.0145328;
   t1[21277] := 0.0147062;
   t1[21278] := 0.014107;
   t1[21279] := 0.0128133;
   t1[21280] := 0.0109134;
   t1[21281] := 0.0084953;
   t1[21282] := 0.005647;
   t1[21283] := 0.0024567;
   t1[21284] := -0.0009876;
   t1[21285] := -0.0045978;
   t1[21286] := -0.0082858;
   t1[21287] := -0.0119636;
   t1[21288] := -0.015543;
   t1[21289] := -0.0189361;
   t1[21290] := -0.0220546;
   t1[21291] := -0.0248106;
   t1[21292] := -0.027116;
   t1[21293] := -0.0288826;
   t1[21294] := -0.0300225;
   t1[21295] := -0.0304475;
   t1[21296] := -0.0300695;
   t1[21297] := -0.0288275;
   t1[21298] := -0.026795;
   t1[21299] := -0.0240877;
   t1[21300] := -0.0279364;
   t1[21301] := -0.032929;
   t1[21302] := -0.0377003;
   t1[21303] := -0.0422051;
   t1[21304] := -0.0463983;
   t1[21305] := -0.0502349;
   t1[21306] := -0.0536697;
   t1[21307] := -0.0566576;
   t1[21308] := -0.0591549;
   t1[21309] := -0.0611399;
   t1[21310] := -0.0626079;
   t1[21311] := -0.063555;
   t1[21312] := -0.0639769;
   t1[21313] := -0.0638697;
   t1[21314] := -0.0632291;
   t1[21315] := -0.0620512;
   t1[21316] := -0.0603318;
   t1[21317] := -0.0580669;
   t1[21318] := -0.0552522;
   t1[21319] := -0.0518839;
   t1[21320] := -0.0479577;
   t1[21321] := -0.0434695;
   t1[21322] := -0.0384153;
   t1[21323] := -0.032791;
   t1[21324] := -0.0265925;
   t1[21325] := -0.0198157;
   t1[21326] := -0.0124565;
   t1[21327] := -0.0045109;
   t1[21328] := 0.0040068;
   t1[21329] := 0.0130485;
   t1[21330] := 0.022562;
   t1[21331] := 0.0324952;
   t1[21332] := 0.0427959;
   t1[21333] := 0.053412;
   t1[21334] := 0.0642915;
   t1[21335] := 0.0753821;
   t1[21336] := 0.0866318;
   t1[21337] := 0.0979884;
   t1[21338] := 0.1093999;
   t1[21339] := 0.1208141;
   t1[21340] := 0.1321788;
   t1[21341] := 0.1434419;
   t1[21342] := 0.1545514;
   t1[21343] := 0.1654552;
   t1[21344] := 0.176101;
   t1[21345] := 0.1864367;
   t1[21346] := 0.1964103;
   t1[21347] := 0.2059735;
   t1[21348] := 0.2150975;
   t1[21349] := 0.2237596;
   t1[21350] := -0.0601228;
   t1[21351] := -0.0677119;
   t1[21352] := -0.0745691;
   t1[21353] := -0.0805743;
   t1[21354] := -0.0856075;
   t1[21355] := -0.0895484;
   t1[21356] := -0.0922769;
   t1[21357] := -0.0936729;
   t1[21358] := -0.0936244;
   t1[21359] := -0.0921452;
   t1[21360] := -0.0893479;
   t1[21361] := -0.0853481;
   t1[21362] := -0.0802611;
   t1[21363] := -0.0742025;
   t1[21364] := -0.0672874;
   t1[21365] := -0.0596316;
   t1[21366] := -0.0513502;
   t1[21367] := -0.0425589;
   t1[21368] := -0.0333729;
   t1[21369] := -0.0239078;
   t1[21370] := -0.0142789;
   t1[21371] := -0.0046016;
   t1[21372] := 0.0050085;
   t1[21373] := 0.0144361;
   t1[21374] := 0.0235658;
   t1[21375] := 0.0322821;
   t1[21376] := 0.0404696;
   t1[21377] := 0.0480134;
   t1[21378] := 0.0548454;
   t1[21379] := 0.0609871;
   t1[21380] := 0.06647;
   t1[21381] := 0.0713255;
   t1[21382] := 0.0755848;
   t1[21383] := 0.0792795;
   t1[21384] := 0.0824409;
   t1[21385] := 0.0851004;
   t1[21386] := 0.0872894;
   t1[21387] := 0.0890393;
   t1[21388] := 0.0903815;
   t1[21389] := 0.0913474;
   t1[21390] := 0.0919683;
   t1[21391] := 0.0922758;
   t1[21392] := 0.0923011;
   t1[21393] := 0.0920758;
   t1[21394] := 0.0916311;
   t1[21395] := 0.0909984;
   t1[21396] := 0.0902092;
   t1[21397] := 0.0892917;
   t1[21398] := 0.0882578;
   t1[21399] := 0.0871147;
   t1[21400] := -0.0200038;
   t1[21401] := -0.0247517;
   t1[21402] := -0.029179;
   t1[21403] := -0.0332124;
   t1[21404] := -0.0367783;
   t1[21405] := -0.0398032;
   t1[21406] := -0.0422137;
   t1[21407] := -0.0439363;
   t1[21408] := -0.0449024;
   t1[21409] := -0.0451195;
   t1[21410] := -0.0446546;
   t1[21411] := -0.0435767;
   t1[21412] := -0.0419546;
   t1[21413] := -0.039857;
   t1[21414] := -0.0373529;
   t1[21415] := -0.0345111;
   t1[21416] := -0.0314003;
   t1[21417] := -0.0280894;
   t1[21418] := -0.0246472;
   t1[21419] := -0.0211426;
   t1[21420] := -0.0176443;
   t1[21421] := -0.0142212;
   t1[21422] := -0.0109422;
   t1[21423] := -0.007876;
   t1[21424] := -0.0050914;
   t1[21425] := -0.0026573;
   t1[21426] := -0.0006426;
   t1[21427] := 0.0008843;
   t1[21428] := 0.0018905;
   t1[21429] := 0.0024104;
   t1[21430] := 0.0024862;
   t1[21431] := 0.0021599;
   t1[21432] := 0.0014734;
   t1[21433] := 0.000469;
   t1[21434] := -0.0008114;
   t1[21435] := -0.0023258;
   t1[21436] := -0.004032;
   t1[21437] := -0.005888;
   t1[21438] := -0.0078518;
   t1[21439] := -0.0098813;
   t1[21440] := -0.0119345;
   t1[21441] := -0.0139692;
   t1[21442] := -0.0159436;
   t1[21443] := -0.0178154;
   t1[21444] := -0.0195427;
   t1[21445] := -0.0210834;
   t1[21446] := -0.0223955;
   t1[21447] := -0.023443;
   t1[21448] := -0.0242204;
   t1[21449] := -0.0247319;
   t1[21450] := 0.0827025;
   t1[21451] := 0.0828631;
   t1[21452] := 0.0828845;
   t1[21453] := 0.0827986;
   t1[21454] := 0.0826372;
   t1[21455] := 0.0824322;
   t1[21456] := 0.0822156;
   t1[21457] := 0.082019;
   t1[21458] := 0.0818736;
   t1[21459] := 0.0817958;
   t1[21460] := 0.081791;
   t1[21461] := 0.0818641;
   t1[21462] := 0.08202;
   t1[21463] := 0.0822638;
   t1[21464] := 0.0826003;
   t1[21465] := 0.0830346;
   t1[21466] := 0.0835717;
   t1[21467] := 0.0842164;
   t1[21468] := 0.0849737;
   t1[21469] := 0.0858486;
   t1[21470] := 0.0868461;
   t1[21471] := 0.0879711;
   t1[21472] := 0.0892287;
   t1[21473] := 0.0906236;
   t1[21474] := 0.092161;
   t1[21475] := 0.0938457;
   t1[21476] := 0.0956828;
   t1[21477] := 0.0976771;
   t1[21478] := 0.0998287;
   t1[21479] := 0.1021284;
   t1[21480] := 0.1045658;
   t1[21481] := 0.1071307;
   t1[21482] := 0.1098129;
   t1[21483] := 0.1126021;
   t1[21484] := 0.1154879;
   t1[21485] := 0.1184602;
   t1[21486] := 0.1215086;
   t1[21487] := 0.124623;
   t1[21488] := 0.1277929;
   t1[21489] := 0.1310082;
   t1[21490] := 0.1342586;
   t1[21491] := 0.1375337;
   t1[21492] := 0.1408234;
   t1[21493] := 0.1441174;
   t1[21494] := 0.1474054;
   t1[21495] := 0.150677;
   t1[21496] := 0.1539222;
   t1[21497] := 0.157128;
   t1[21498] := 0.1602693;
   t1[21499] := 0.163317;
   t1[21500] := -0.2512962;
   t1[21501] := -0.2436767;
   t1[21502] := -0.2353746;
   t1[21503] := -0.2263576;
   t1[21504] := -0.2165938;
   t1[21505] := -0.2060509;
   t1[21506] := -0.1946967;
   t1[21507] := -0.1824992;
   t1[21508] := -0.1694303;
   t1[21509] := -0.1555257;
   t1[21510] := -0.1408714;
   t1[21511] := -0.1255546;
   t1[21512] := -0.1096625;
   t1[21513] := -0.0932824;
   t1[21514] := -0.0765017;
   t1[21515] := -0.0594074;
   t1[21516] := -0.042087;
   t1[21517] := -0.0246276;
   t1[21518] := -0.0071165;
   t1[21519] := 0.010359;
   t1[21520] := 0.0277116;
   t1[21521] := 0.0448542;
   t1[21522] := 0.0616994;
   t1[21523] := 0.07816;
   t1[21524] := 0.0941487;
   t1[21525] := 0.1095782;
   t1[21526] := 0.1243613;
   t1[21527] := 0.1384111;
   t1[21528] := 0.1516734;
   t1[21529] := 0.1641564;
   t1[21530] := 0.1758753;
   t1[21531] := 0.186845;
   t1[21532] := 0.1970809;
   t1[21533] := 0.2065979;
   t1[21534] := 0.2154113;
   t1[21535] := 0.2235361;
   t1[21536] := 0.2309875;
   t1[21537] := 0.2377806;
   t1[21538] := 0.2439306;
   t1[21539] := 0.2494525;
   t1[21540] := 0.2543615;
   t1[21541] := 0.2586727;
   t1[21542] := 0.2624012;
   t1[21543] := 0.2655622;
   t1[21544] := 0.2681709;
   t1[21545] := 0.2702422;
   t1[21546] := 0.2717913;
   t1[21547] := 0.2728322;
   t1[21548] := 0.2733715;
   t1[21549] := 0.2734144;
   t1[21550] := -0.1341166;
   t1[21551] := -0.129175;
   t1[21552] := -0.1240045;
   t1[21553] := -0.1186445;
   t1[21554] := -0.1131344;
   t1[21555] := -0.1075137;
   t1[21556] := -0.1018216;
   t1[21557] := -0.0960976;
   t1[21558] := -0.0903789;
   t1[21559] := -0.0846687;
   t1[21560] := -0.0789433;
   t1[21561] := -0.0731783;
   t1[21562] := -0.0673495;
   t1[21563] := -0.0614326;
   t1[21564] := -0.0554031;
   t1[21565] := -0.0492367;
   t1[21566] := -0.0429091;
   t1[21567] := -0.036396;
   t1[21568] := -0.0296731;
   t1[21569] := -0.0227159;
   t1[21570] := -0.0155001;
   t1[21571] := -0.0080015;
   t1[21572] := -0.0001956;
   t1[21573] := 0.0079418;
   t1[21574] := 0.0164352;
   t1[21575] := 0.0253088;
   t1[21576] := 0.0345869;
   t1[21577] := 0.0442938;
   t1[21578] := 0.0544231;
   t1[21579] := 0.0649119;
   t1[21580] := 0.0756905;
   t1[21581] := 0.0866892;
   t1[21582] := 0.0978385;
   t1[21583] := 0.1090688;
   t1[21584] := 0.1203106;
   t1[21585] := 0.1314942;
   t1[21586] := 0.14255;
   t1[21587] := 0.1534084;
   t1[21588] := 0.1639999;
   t1[21589] := 0.1742549;
   t1[21590] := 0.1841038;
   t1[21591] := 0.1934769;
   t1[21592] := 0.2023047;
   t1[21593] := 0.2105176;
   t1[21594] := 0.2180461;
   t1[21595] := 0.2248204;
   t1[21596] := 0.2307711;
   t1[21597] := 0.2358411;
   t1[21598] := 0.2400362;
   t1[21599] := 0.2433818;
   t1[21600] := -0.1029919;
   t1[21601] := -0.0909107;
   t1[21602] := -0.0791188;
   t1[21603] := -0.0677159;
   t1[21604] := -0.0568019;
   t1[21605] := -0.0464767;
   t1[21606] := -0.03684;
   t1[21607] := -0.0279917;
   t1[21608] := -0.0200273;
   t1[21609] := -0.0129723;
   t1[21610] := -0.0067978;
   t1[21611] := -0.0014734;
   t1[21612] := 0.0030316;
   t1[21613] := 0.0067475;
   t1[21614] := 0.0097049;
   t1[21615] := 0.0119343;
   t1[21616] := 0.0134661;
   t1[21617] := 0.0143308;
   t1[21618] := 0.0145591;
   t1[21619] := 0.0141812;
   t1[21620] := 0.0132278;
   t1[21621] := 0.0117293;
   t1[21622] := 0.0097162;
   t1[21623] := 0.007219;
   t1[21624] := 0.0042682;
   t1[21625] := 0.0008943;
   t1[21626] := -0.0028722;
   t1[21627] := -0.0070008;
   t1[21628] := -0.0114623;
   t1[21629] := -0.0162299;
   t1[21630] := -0.0212768;
   t1[21631] := -0.0265765;
   t1[21632] := -0.0321023;
   t1[21633] := -0.0378277;
   t1[21634] := -0.043726;
   t1[21635] := -0.0497706;
   t1[21636] := -0.0559349;
   t1[21637] := -0.0621922;
   t1[21638] := -0.068516;
   t1[21639] := -0.0748796;
   t1[21640] := -0.0812563;
   t1[21641] := -0.0876197;
   t1[21642] := -0.093943;
   t1[21643] := -0.1001997;
   t1[21644] := -0.1063631;
   t1[21645] := -0.1124066;
   t1[21646] := -0.1183036;
   t1[21647] := -0.124028;
   t1[21648] := -0.1295565;
   t1[21649] := -0.1348667;
   t1[21650] := -0.0090596;
   t1[21651] := -0.00353;
   t1[21652] := 0.0015623;
   t1[21653] := 0.0061335;
   t1[21654] := 0.0101;
   t1[21655] := 0.013378;
   t1[21656] := 0.0158839;
   t1[21657] := 0.017534;
   t1[21658] := 0.0182505;
   t1[21659] := 0.0180475;
   t1[21660] := 0.0170114;
   t1[21661] := 0.0152307;
   t1[21662] := 0.0127936;
   t1[21663] := 0.0097885;
   t1[21664] := 0.0063039;
   t1[21665] := 0.002428;
   t1[21666] := -0.0017508;
   t1[21667] := -0.0061441;
   t1[21668] := -0.0106635;
   t1[21669] := -0.0152208;
   t1[21670] := -0.0197274;
   t1[21671] := -0.0240951;
   t1[21672] := -0.0282355;
   t1[21673] := -0.0320603;
   t1[21674] := -0.035481;
   t1[21675] := -0.0384092;
   t1[21676] := -0.0407568;
   t1[21677] := -0.0424356;
   t1[21678] := -0.0434054;
   t1[21679] := -0.0437158;
   t1[21680] := -0.0434269;
   t1[21681] := -0.0425985;
   t1[21682] := -0.0412905;
   t1[21683] := -0.0395627;
   t1[21684] := -0.037475;
   t1[21685] := -0.0350874;
   t1[21686] := -0.0324596;
   t1[21687] := -0.0296516;
   t1[21688] := -0.0267231;
   t1[21689] := -0.0237342;
   t1[21690] := -0.0207447;
   t1[21691] := -0.0178145;
   t1[21692] := -0.0150034;
   t1[21693] := -0.0123713;
   t1[21694] := -0.0099781;
   t1[21695] := -0.0078837;
   t1[21696] := -0.0061479;
   t1[21697] := -0.0048187;
   t1[21698] := -0.0038843;
   t1[21699] := -0.0033141;
   t1[21700] := -0.192581;
   t1[21701] := -0.1813929;
   t1[21702] := -0.170114;
   t1[21703] := -0.1588169;
   t1[21704] := -0.1475747;
   t1[21705] := -0.1364602;
   t1[21706] := -0.1255462;
   t1[21707] := -0.1149055;
   t1[21708] := -0.1046085;
   t1[21709] := -0.0946843;
   t1[21710] := -0.0851298;
   t1[21711] := -0.0759411;
   t1[21712] := -0.0671143;
   t1[21713] := -0.0586454;
   t1[21714] := -0.0505305;
   t1[21715] := -0.0427657;
   t1[21716] := -0.035347;
   t1[21717] := -0.0282705;
   t1[21718] := -0.0215323;
   t1[21719] := -0.0151285;
   t1[21720] := -0.009055;
   t1[21721] := -0.003308;
   t1[21722] := 0.0021165;
   t1[21723] := 0.0072223;
   t1[21724] := 0.0120135;
   t1[21725] := 0.016494;
   t1[21726] := 0.0206677;
   t1[21727] := 0.0245385;
   t1[21728] := 0.0281083;
   t1[21729] := 0.0313753;
   t1[21730] := 0.0343374;
   t1[21731] := 0.0369921;
   t1[21732] := 0.0393372;
   t1[21733] := 0.0413706;
   t1[21734] := 0.0430899;
   t1[21735] := 0.0444928;
   t1[21736] := 0.0455772;
   t1[21737] := 0.0463408;
   t1[21738] := 0.0467813;
   t1[21739] := 0.0468964;
   t1[21740] := 0.046684;
   t1[21741] := 0.0461417;
   t1[21742] := 0.0452672;
   t1[21743] := 0.0440585;
   t1[21744] := 0.0425131;
   t1[21745] := 0.0406288;
   t1[21746] := 0.0384034;
   t1[21747] := 0.0358393;
   t1[21748] := 0.0329625;
   t1[21749] := 0.0298061;
   t1[21750] := 0.1197442;
   t1[21751] := 0.1263732;
   t1[21752] := 0.1331062;
   t1[21753] := 0.1399399;
   t1[21754] := 0.1468707;
   t1[21755] := 0.1538952;
   t1[21756] := 0.1610098;
   t1[21757] := 0.1682112;
   t1[21758] := 0.1754922;
   t1[21759] := 0.1827909;
   t1[21760] := 0.1900021;
   t1[21761] := 0.1970194;
   t1[21762] := 0.2037365;
   t1[21763] := 0.210047;
   t1[21764] := 0.2158445;
   t1[21765] := 0.2210227;
   t1[21766] := 0.2254753;
   t1[21767] := 0.2290957;
   t1[21768] := 0.2317777;
   t1[21769] := 0.2334149;
   t1[21770] := 0.2339009;
   t1[21771] := 0.2331294;
   t1[21772] := 0.230994;
   t1[21773] := 0.2273884;
   t1[21774] := 0.2222061;
   t1[21775] := 0.2153407;
   t1[21776] := 0.2066861;
   t1[21777] := 0.1961366;
   t1[21778] := 0.1836909;
   t1[21779] := 0.1695445;
   t1[21780] := 0.153915;
   t1[21781] := 0.1370202;
   t1[21782] := 0.1190776;
   t1[21783] := 0.1003049;
   t1[21784] := 0.0809195;
   t1[21785] := 0.0611394;
   t1[21786] := 0.041182;
   t1[21787] := 0.0212649;
   t1[21788] := 0.0016058;
   t1[21789] := -0.0175778;
   t1[21790] := -0.036068;
   t1[21791] := -0.0536474;
   t1[21792] := -0.0700983;
   t1[21793] := -0.0852031;
   t1[21794] := -0.0987442;
   t1[21795] := -0.1105038;
   t1[21796] := -0.1202645;
   t1[21797] := -0.1278576;
   t1[21798] := -0.13336;
   t1[21799] := -0.1369247;
   t1[21800] := 0.1101966;
   t1[21801] := 0.1051921;
   t1[21802] := 0.0997305;
   t1[21803] := 0.093831;
   t1[21804] := 0.0875128;
   t1[21805] := 0.0807951;
   t1[21806] := 0.073697;
   t1[21807] := 0.0662378;
   t1[21808] := 0.0584364;
   t1[21809] := 0.0503086;
   t1[21810] := 0.0418673;
   t1[21811] := 0.0331255;
   t1[21812] := 0.0240962;
   t1[21813] := 0.0147923;
   t1[21814] := 0.0052269;
   t1[21815] := -0.004587;
   t1[21816] := -0.0146366;
   t1[21817] := -0.0249088;
   t1[21818] := -0.0353906;
   t1[21819] := -0.0460691;
   t1[21820] := -0.0569313;
   t1[21821] := -0.0679642;
   t1[21822] := -0.0791548;
   t1[21823] := -0.0904902;
   t1[21824] := -0.1019574;
   t1[21825] := -0.1135434;
   t1[21826] := -0.1252352;
   t1[21827] := -0.1370196;
   t1[21828] := -0.1488545;
   t1[21829] := -0.1606431;
   t1[21830] := -0.1722825;
   t1[21831] := -0.1836698;
   t1[21832] := -0.194702;
   t1[21833] := -0.2052764;
   t1[21834] := -0.2152898;
   t1[21835] := -0.2246395;
   t1[21836] := -0.2332225;
   t1[21837] := -0.240936;
   t1[21838] := -0.2476769;
   t1[21839] := -0.2533424;
   t1[21840] := -0.2578297;
   t1[21841] := -0.2610357;
   t1[21842] := -0.2628575;
   t1[21843] := -0.2631924;
   t1[21844] := -0.2619372;
   t1[21845] := -0.2589892;
   t1[21846] := -0.2542455;
   t1[21847] := -0.2476377;
   t1[21848] := -0.2392711;
   t1[21849] := -0.2293047;
   t1[21850] := -0.2120533;
   t1[21851] := -0.2008377;
   t1[21852] := -0.1895115;
   t1[21853] := -0.1781628;
   t1[21854] := -0.1668795;
   t1[21855] := -0.1557498;
   t1[21856] := -0.1448617;
   t1[21857] := -0.1343032;
   t1[21858] := -0.1241578;
   t1[21859] := -0.1144379;
   t1[21860] := -0.1050999;
   t1[21861] := -0.0960986;
   t1[21862] := -0.0873888;
   t1[21863] := -0.0789256;
   t1[21864] := -0.0706636;
   t1[21865] := -0.0625579;
   t1[21866] := -0.0545633;
   t1[21867] := -0.0466346;
   t1[21868] := -0.0387267;
   t1[21869] := -0.0307946;
   t1[21870] := -0.022793;
   t1[21871] := -0.0146768;
   t1[21872] := -0.006401;
   t1[21873] := 0.0020797;
   t1[21874] := 0.0108103;
   t1[21875] := 0.019836;
   t1[21876] := 0.0292019;
   t1[21877] := 0.0389526;
   t1[21878] := 0.0490809;
   t1[21879] := 0.0594808;
   t1[21880] := 0.0700353;
   t1[21881] := 0.0806274;
   t1[21882] := 0.0911404;
   t1[21883] := 0.1014571;
   t1[21884] := 0.1114607;
   t1[21885] := 0.1210342;
   t1[21886] := 0.1300607;
   t1[21887] := 0.1384232;
   t1[21888] := 0.1460048;
   t1[21889] := 0.1526886;
   t1[21890] := 0.1583575;
   t1[21891] := 0.1628947;
   t1[21892] := 0.1661831;
   t1[21893] := 0.168106;
   t1[21894] := 0.1685463;
   t1[21895] := 0.167387;
   t1[21896] := 0.1645113;
   t1[21897] := 0.1598403;
   t1[21898] := 0.1534863;
   t1[21899] := 0.1456208;
   t1[21900] := 0.0065645;
   t1[21901] := 0.0131053;
   t1[21902] := 0.0188022;
   t1[21903] := 0.0235609;
   t1[21904] := 0.0272877;
   t1[21905] := 0.0298884;
   t1[21906] := 0.0312691;
   t1[21907] := 0.0313356;
   t1[21908] := 0.0300022;
   t1[21909] := 0.0273089;
   t1[21910] := 0.0233949;
   t1[21911] := 0.018402;
   t1[21912] := 0.0124722;
   t1[21913] := 0.0057472;
   t1[21914] := -0.001631;
   t1[21915] := -0.0095206;
   t1[21916] := -0.0177797;
   t1[21917] := -0.0262665;
   t1[21918] := -0.034839;
   t1[21919] := -0.0433554;
   t1[21920] := -0.0516739;
   t1[21921] := -0.0596525;
   t1[21922] := -0.0671494;
   t1[21923] := -0.0740228;
   t1[21924] := -0.0801307;
   t1[21925] := -0.0853314;
   t1[21926] := -0.0894828;
   t1[21927] := -0.0924439;
   t1[21928] := -0.0941494;
   t1[21929] := -0.094678;
   t1[21930] := -0.0941246;
   t1[21931] := -0.092584;
   t1[21932] := -0.0901509;
   t1[21933] := -0.0869202;
   t1[21934] := -0.0829866;
   t1[21935] := -0.0784451;
   t1[21936] := -0.0733904;
   t1[21937] := -0.0679173;
   t1[21938] := -0.0621206;
   t1[21939] := -0.0560952;
   t1[21940] := -0.0499358;
   t1[21941] := -0.0437373;
   t1[21942] := -0.0375945;
   t1[21943] := -0.0316022;
   t1[21944] := -0.0258552;
   t1[21945] := -0.0204482;
   t1[21946] := -0.0154762;
   t1[21947] := -0.0110187;
   t1[21948] := -0.0070789;
   t1[21949] := -0.0036363;
   t1[21950] := -0.1478585;
   t1[21951] := -0.1349572;
   t1[21952] := -0.1218061;
   t1[21953] := -0.1084367;
   t1[21954] := -0.0948808;
   t1[21955] := -0.0811699;
   t1[21956] := -0.0673356;
   t1[21957] := -0.0534096;
   t1[21958] := -0.0394242;
   t1[21959] := -0.0254223;
   t1[21960] := -0.0114554;
   t1[21961] := 0.0024249;
   t1[21962] := 0.016167;
   t1[21963] := 0.0297191;
   t1[21964] := 0.0430296;
   t1[21965] := 0.056047;
   t1[21966] := 0.0687196;
   t1[21967] := 0.0809956;
   t1[21968] := 0.0928236;
   t1[21969] := 0.1041518;
   t1[21970] := 0.1149286;
   t1[21971] := 0.1251023;
   t1[21972] := 0.1346213;
   t1[21973] := 0.143434;
   t1[21974] := 0.1514887;
   t1[21975] := 0.1587338;
   t1[21976] := 0.1651177;
   t1[21977] := 0.1705888;
   t1[21978] := 0.1751249;
   t1[21979] := 0.1787581;
   t1[21980] := 0.1815271;
   t1[21981] := 0.18347;
   t1[21982] := 0.1846256;
   t1[21983] := 0.1850321;
   t1[21984] := 0.184728;
   t1[21985] := 0.1837518;
   t1[21986] := 0.182142;
   t1[21987] := 0.1799369;
   t1[21988] := 0.177175;
   t1[21989] := 0.1738947;
   t1[21990] := 0.1701346;
   t1[21991] := 0.165933;
   t1[21992] := 0.1613284;
   t1[21993] := 0.1563593;
   t1[21994] := 0.151064;
   t1[21995] := 0.1454811;
   t1[21996] := 0.1396489;
   t1[21997] := 0.133602;
   t1[21998] := 0.1273545;
   t1[21999] := 0.1209146;
   t1[22000] := 0.1370825;
   t1[22001] := 0.1391352;
   t1[22002] := 0.1407191;
   t1[22003] := 0.1417688;
   t1[22004] := 0.142219;
   t1[22005] := 0.1420043;
   t1[22006] := 0.1410592;
   t1[22007] := 0.1393185;
   t1[22008] := 0.1367226;
   t1[22009] := 0.1333001;
   t1[22010] := 0.1291494;
   t1[22011] := 0.1243709;
   t1[22012] := 0.1190648;
   t1[22013] := 0.1133314;
   t1[22014] := 0.1072708;
   t1[22015] := 0.1009835;
   t1[22016] := 0.0945697;
   t1[22017] := 0.0881296;
   t1[22018] := 0.0817635;
   t1[22019] := 0.0755717;
   t1[22020] := 0.0696544;
   t1[22021] := 0.064112;
   t1[22022] := 0.0590446;
   t1[22023] := 0.0545525;
   t1[22024] := 0.0507361;
   t1[22025] := 0.0476955;
   t1[22026] := 0.0455311;
   t1[22027] := 0.0443425;
   t1[22028] := 0.044159;
   t1[22029] := 0.0448768;
   t1[22030] := 0.0463771;
   t1[22031] := 0.048541;
   t1[22032] := 0.0512499;
   t1[22033] := 0.054385;
   t1[22034] := 0.0578275;
   t1[22035] := 0.0614587;
   t1[22036] := 0.0651597;
   t1[22037] := 0.0688118;
   t1[22038] := 0.0722963;
   t1[22039] := 0.0754943;
   t1[22040] := 0.0782871;
   t1[22041] := 0.080556;
   t1[22042] := 0.0821821;
   t1[22043] := 0.0830467;
   t1[22044] := 0.0830311;
   t1[22045] := 0.0820164;
   t1[22046] := 0.0798839;
   t1[22047] := 0.0765467;
   t1[22048] := 0.0720777;
   t1[22049] := 0.0665991;
   t1[22050] := 0.1807702;
   t1[22051] := 0.1741173;
   t1[22052] := 0.1672406;
   t1[22053] := 0.1601745;
   t1[22054] := 0.1529535;
   t1[22055] := 0.1456123;
   t1[22056] := 0.1381852;
   t1[22057] := 0.130707;
   t1[22058] := 0.123212;
   t1[22059] := 0.1157338;
   t1[22060] := 0.1083055;
   t1[22061] := 0.10096;
   t1[22062] := 0.0937301;
   t1[22063] := 0.0866489;
   t1[22064] := 0.0797492;
   t1[22065] := 0.0730641;
   t1[22066] := 0.0666263;
   t1[22067] := 0.060469;
   t1[22068] := 0.0546249;
   t1[22069] := 0.0491271;
   t1[22070] := 0.0440085;
   t1[22071] := 0.0393019;
   t1[22072] := 0.0350404;
   t1[22073] := 0.0312569;
   t1[22074] := 0.0279843;
   t1[22075] := 0.0252555;
   t1[22076] := 0.0231035;
   t1[22077] := 0.0215609;
   t1[22078] := 0.0206299;
   t1[22079] := 0.0202547;
   t1[22080] := 0.0203728;
   t1[22081] := 0.0209221;
   t1[22082] := 0.0218403;
   t1[22083] := 0.0230651;
   t1[22084] := 0.0245342;
   t1[22085] := 0.0261853;
   t1[22086] := 0.0279561;
   t1[22087] := 0.0297844;
   t1[22088] := 0.0316078;
   t1[22089] := 0.0333641;
   t1[22090] := 0.034991;
   t1[22091] := 0.0364261;
   t1[22092] := 0.0376073;
   t1[22093] := 0.0384723;
   t1[22094] := 0.0389587;
   t1[22095] := 0.0390042;
   t1[22096] := 0.0385466;
   t1[22097] := 0.0375389;
   t1[22098] := 0.0360107;
   t1[22099] := 0.0340154;
   t1[22100] := 0.1694753;
   t1[22101] := 0.1553752;
   t1[22102] := 0.1413849;
   t1[22103] := 0.1276387;
   t1[22104] := 0.1142712;
   t1[22105] := 0.1014168;
   t1[22106] := 0.0892098;
   t1[22107] := 0.0777849;
   t1[22108] := 0.0672688;
   t1[22109] := 0.0576726;
   t1[22110] := 0.0489159;
   t1[22111] := 0.0409158;
   t1[22112] := 0.0335895;
   t1[22113] := 0.0268542;
   t1[22114] := 0.0206269;
   t1[22115] := 0.014825;
   t1[22116] := 0.0093655;
   t1[22117] := 0.0041656;
   t1[22118] := -0.0008576;
   t1[22119] := -0.0057869;
   t1[22120] := -0.010705;
   t1[22121] := -0.015695;
   t1[22122] := -0.0208395;
   t1[22123] := -0.0262215;
   t1[22124] := -0.0319237;
   t1[22125] := -0.0380291;
   t1[22126] := -0.0446204;
   t1[22127] := -0.05178;
   t1[22128] := -0.0595318;
   t1[22129] := -0.0677888;
   t1[22130] := -0.0764519;
   t1[22131] := -0.0854217;
   t1[22132] := -0.094599;
   t1[22133] := -0.1038845;
   t1[22134] := -0.113179;
   t1[22135] := -0.1223832;
   t1[22136] := -0.1313979;
   t1[22137] := -0.1401237;
   t1[22138] := -0.1484615;
   t1[22139] := -0.156312;
   t1[22140] := -0.1635759;
   t1[22141] := -0.1701539;
   t1[22142] := -0.1759469;
   t1[22143] := -0.1808555;
   t1[22144] := -0.1847805;
   t1[22145] := -0.1876225;
   t1[22146] := -0.1892825;
   t1[22147] := -0.1896862;
   t1[22148] := -0.1888851;
   t1[22149] := -0.1869699;
   t1[22150] := 0.1395302;
   t1[22151] := 0.1385239;
   t1[22152] := 0.1373932;
   t1[22153] := 0.1361011;
   t1[22154] := 0.1346105;
   t1[22155] := 0.1328844;
   t1[22156] := 0.1308859;
   t1[22157] := 0.1285779;
   t1[22158] := 0.1259261;
   t1[22159] := 0.1229387;
   t1[22160] := 0.1196572;
   t1[22161] := 0.116124;
   t1[22162] := 0.1123814;
   t1[22163] := 0.108472;
   t1[22164] := 0.1044381;
   t1[22165] := 0.1003221;
   t1[22166] := 0.0961664;
   t1[22167] := 0.0920134;
   t1[22168] := 0.0879056;
   t1[22169] := 0.0838853;
   t1[22170] := 0.0799949;
   t1[22171] := 0.0762769;
   t1[22172] := 0.0727736;
   t1[22173] := 0.0695275;
   t1[22174] := 0.0665809;
   t1[22175] := 0.0639763;
   t1[22176] := 0.0617561;
   t1[22177] := 0.0599625;
   t1[22178] := 0.0586142;
   t1[22179] := 0.0576856;
   t1[22180] := 0.0571461;
   t1[22181] := 0.056965;
   t1[22182] := 0.0571119;
   t1[22183] := 0.057556;
   t1[22184] := 0.0582668;
   t1[22185] := 0.0592136;
   t1[22186] := 0.0603659;
   t1[22187] := 0.0616931;
   t1[22188] := 0.0631645;
   t1[22189] := 0.0647496;
   t1[22190] := 0.0664177;
   t1[22191] := 0.0681383;
   t1[22192] := 0.0698806;
   t1[22193] := 0.0716143;
   t1[22194] := 0.0733085;
   t1[22195] := 0.0749328;
   t1[22196] := 0.0764564;
   t1[22197] := 0.0778522;
   t1[22198] := 0.0791089;
   t1[22199] := 0.0802208;
   t1[22200] := 0.1470823;
   t1[22201] := 0.1396195;
   t1[22202] := 0.1314362;
   t1[22203] := 0.1225874;
   t1[22204] := 0.1131281;
   t1[22205] := 0.103113;
   t1[22206] := 0.0925971;
   t1[22207] := 0.0816353;
   t1[22208] := 0.0702827;
   t1[22209] := 0.0585969;
   t1[22210] := 0.0466374;
   t1[22211] := 0.0344639;
   t1[22212] := 0.022136;
   t1[22213] := 0.0097134;
   t1[22214] := -0.0027442;
   t1[22215] := -0.0151773;
   t1[22216] := -0.0275262;
   t1[22217] := -0.0397313;
   t1[22218] := -0.0517329;
   t1[22219] := -0.0634713;
   t1[22220] := -0.074887;
   t1[22221] := -0.0859203;
   t1[22222] := -0.0965115;
   t1[22223] := -0.106601;
   t1[22224] := -0.1161292;
   t1[22225] := -0.1250364;
   t1[22226] := -0.133263;
   t1[22227] := -0.1407496;
   t1[22228] := -0.1474703;
   t1[22229] := -0.1534624;
   t1[22230] := -0.1587702;
   t1[22231] := -0.1634381;
   t1[22232] := -0.1675105;
   t1[22233] := -0.1710317;
   t1[22234] := -0.1740462;
   t1[22235] := -0.1765982;
   t1[22236] := -0.1787322;
   t1[22237] := -0.1804925;
   t1[22238] := -0.1819234;
   t1[22239] := -0.1830695;
   t1[22240] := -0.1839749;
   t1[22241] := -0.1846841;
   t1[22242] := -0.1852415;
   t1[22243] := -0.1856914;
   t1[22244] := -0.1860782;
   t1[22245] := -0.1864462;
   t1[22246] := -0.1868398;
   t1[22247] := -0.1872934;
   t1[22248] := -0.18779;
   t1[22249] := -0.1882973;
   t1[22250] := 0.2214328;
   t1[22251] := 0.2061494;
   t1[22252] := 0.1907533;
   t1[22253] := 0.1753337;
   t1[22254] := 0.1599798;
   t1[22255] := 0.1447807;
   t1[22256] := 0.1298254;
   t1[22257] := 0.1152031;
   t1[22258] := 0.1010003;
   t1[22259] := 0.0872605;
   t1[22260] := 0.0739941;
   t1[22261] := 0.0612103;
   t1[22262] := 0.0489182;
   t1[22263] := 0.0371274;
   t1[22264] := 0.0258469;
   t1[22265] := 0.0150862;
   t1[22266] := 0.0048543;
   t1[22267] := -0.0048392;
   t1[22268] := -0.0139853;
   t1[22269] := -0.0225745;
   t1[22270] := -0.0305977;
   t1[22271] := -0.0380455;
   t1[22272] := -0.0449087;
   t1[22273] := -0.0511779;
   t1[22274] := -0.056844;
   t1[22275] := -0.0618976;
   t1[22276] := -0.0663295;
   t1[22277] := -0.0701305;
   t1[22278] := -0.0733068;
   t1[22279] := -0.0758934;
   t1[22280] := -0.0779286;
   t1[22281] := -0.0794509;
   t1[22282] := -0.0804984;
   t1[22283] := -0.0811096;
   t1[22284] := -0.0813227;
   t1[22285] := -0.081176;
   t1[22286] := -0.080708;
   t1[22287] := -0.0799568;
   t1[22288] := -0.0789609;
   t1[22289] := -0.0777585;
   t1[22290] := -0.076388;
   t1[22291] := -0.0748877;
   t1[22292] := -0.0732959;
   t1[22293] := -0.0716509;
   t1[22294] := -0.0699911;
   t1[22295] := -0.0683548;
   t1[22296] := -0.0667802;
   t1[22297] := -0.0652994;
   t1[22298] := -0.0639122;
   t1[22299] := -0.0626088;
   t1[22300] := 0.123815;
   t1[22301] := 0.1239887;
   t1[22302] := 0.1236951;
   t1[22303] := 0.1229381;
   t1[22304] := 0.1217219;
   t1[22305] := 0.1200506;
   t1[22306] := 0.1179283;
   t1[22307] := 0.1153592;
   t1[22308] := 0.1123488;
   t1[22309] := 0.1089228;
   t1[22310] := 0.1051236;
   t1[22311] := 0.1009937;
   t1[22312] := 0.0965755;
   t1[22313] := 0.0919118;
   t1[22314] := 0.0870451;
   t1[22315] := 0.0820179;
   t1[22316] := 0.0768728;
   t1[22317] := 0.0716523;
   t1[22318] := 0.0663991;
   t1[22319] := 0.0611557;
   t1[22320] := 0.0559647;
   t1[22321] := 0.0508686;
   t1[22322] := 0.04591;
   t1[22323] := 0.0411315;
   t1[22324] := 0.0365755;
   t1[22325] := 0.0322848;
   t1[22326] := 0.0283019;
   t1[22327] := 0.0246691;
   t1[22328] := 0.0214091;
   t1[22329] := 0.0185071;
   t1[22330] := 0.015944;
   t1[22331] := 0.0137009;
   t1[22332] := 0.0117588;
   t1[22333] := 0.0100986;
   t1[22334] := 0.0087013;
   t1[22335] := 0.007548;
   t1[22336] := 0.0066197;
   t1[22337] := 0.0058973;
   t1[22338] := 0.0053618;
   t1[22339] := 0.0049943;
   t1[22340] := 0.0047757;
   t1[22341] := 0.004687;
   t1[22342] := 0.0047093;
   t1[22343] := 0.0048234;
   t1[22344] := 0.0050105;
   t1[22345] := 0.0052516;
   t1[22346] := 0.0055275;
   t1[22347] := 0.0058216;
   t1[22348] := 0.006128;
   t1[22349] := 0.0064445;
   t1[22350] := 0.3236379;
   t1[22351] := 0.3133089;
   t1[22352] := 0.3023048;
   t1[22353] := 0.2906519;
   t1[22354] := 0.2783762;
   t1[22355] := 0.2655037;
   t1[22356] := 0.2520607;
   t1[22357] := 0.2380731;
   t1[22358] := 0.2235684;
   t1[22359] := 0.2085918;
   t1[22360] := 0.1932031;
   t1[22361] := 0.1774625;
   t1[22362] := 0.1614299;
   t1[22363] := 0.1451657;
   t1[22364] := 0.1287298;
   t1[22365] := 0.1121823;
   t1[22366] := 0.0955834;
   t1[22367] := 0.0789932;
   t1[22368] := 0.0624718;
   t1[22369] := 0.0460793;
   t1[22370] := 0.0298759;
   t1[22371] := 0.0139215;
   t1[22372] := -0.0017236;
   t1[22373] := -0.0169994;
   t1[22374] := -0.0318458;
   t1[22375] := -0.0462025;
